C03647=1188.648,139.249,-53.696,-178.416,6.243,148.660
C03648=1188.653,139.000,-53.675,-178.419,6.241,148.660
C03649=1188.658,138.751,-53.655,-178.422,6.239,148.661
C03650=1188.662,138.502,-53.634,-178.424,6.238,148.661
C03651=1188.667,138.252,-53.615,-178.427,6.237,148.662
C03652=1188.672,138.003,-53.594,-178.430,6.235,148.662
C03653=1188.676,137.754,-53.573,-178.432,6.233,148.663
C03654=1188.681,137.505,-53.553,-178.435,6.232,148.663
C03655=1188.686,137.256,-53.532,-178.438,6.231,148.664
C03656=1188.691,137.006,-53.512,-178.440,6.229,148.664
C03657=1188.696,136.758,-53.492,-178.443,6.227,148.664
C03658=1188.700,136.509,-53.472,-178.445,6.226,148.665
C03659=1188.705,136.260,-53.451,-178.448,6.225,148.665
C03660=1188.710,136.010,-53.431,-178.451,6.223,148.666
C03661=1188.714,135.761,-53.411,-178.453,6.222,148.666
C03662=1188.719,135.512,-53.390,-178.456,6.220,148.667
C03663=1188.724,135.262,-53.370,-178.459,6.219,148.667
C03664=1188.729,135.013,-53.350,-178.462,6.217,148.668
C03665=1188.733,134.764,-53.329,-178.464,6.216,148.668
C03666=1188.738,134.515,-53.309,-178.467,6.215,148.668
C03667=1188.744,134.266,-53.289,-178.470,6.213,148.669
C03668=1188.748,134.017,-53.269,-178.472,6.212,148.669
C03669=1188.753,133.768,-53.249,-178.475,6.210,148.670
C03670=1188.757,133.519,-53.229,-178.477,6.209,148.670
C03671=1188.762,133.270,-53.208,-178.480,6.207,148.671
C03672=1188.768,133.001,-53.187,-178.483,6.206,148.671
C03673=1188.772,132.733,-53.165,-178.486,6.205,148.672
C03674=1188.778,132.464,-53.143,-178.488,6.203,148.672
C03675=1188.783,132.195,-53.122,-178.491,6.201,148.673
C03676=1188.787,131.946,-53.102,-178.494,6.200,148.673
C03677=1188.793,131.696,-53.082,-178.497,6.198,148.674
C03678=1188.797,131.447,-53.061,-178.499,6.197,148.674
C03679=1188.802,131.199,-53.042,-178.502,6.196,148.675
C03680=1188.807,130.950,-53.022,-178.505,6.194,148.675
C03681=1188.811,130.701,-53.001,-178.507,6.193,148.675
C03682=1188.816,130.451,-52.981,-178.510,6.191,148.676
C03683=1188.820,130.202,-52.961,-178.513,6.190,148.676
C03684=1188.825,129.953,-52.941,-178.515,6.189,148.677
C03685=1188.831,129.704,-52.922,-178.518,6.187,148.677
C03686=1188.836,129.455,-52.901,-178.521,6.186,148.678
C03687=1188.840,129.205,-52.882,-178.523,6.185,148.678
C03688=1188.845,128.956,-52.861,-178.526,6.183,148.679
C03689=1188.850,128.707,-52.842,-178.529,6.181,148.679
C03690=1188.855,128.458,-52.821,-178.531,6.181,148.680
C03691=1188.859,128.209,-52.802,-178.534,6.179,148.680
C03692=1188.864,127.959,-52.782,-178.537,6.177,148.680
C03693=1188.869,127.710,-52.762,-178.539,6.177,148.681
C03694=1188.874,127.461,-52.743,-178.542,6.175,148.681
C03695=1188.878,127.212,-52.722,-178.545,6.173,148.682
C03696=1188.883,126.963,-52.702,-178.547,6.172,148.682
C03697=1188.888,126.713,-52.683,-178.550,6.171,148.683
C03698=1188.893,126.465,-52.663,-178.553,6.169,148.683
C03699=1188.898,126.215,-52.643,-178.555,6.168,148.684
C03700=1188.902,125.966,-52.624,-178.558,6.167,148.684
C03701=1188.907,125.717,-52.603,-178.561,6.165,148.685
C03702=1188.912,125.468,-52.584,-178.563,6.164,148.685
C03703=1188.916,125.219,-52.565,-178.566,6.163,148.686
C03704=1188.921,124.970,-52.544,-178.569,6.161,148.686
C03705=1188.926,124.721,-52.525,-178.571,6.160,148.686
C03706=1188.931,124.471,-52.505,-178.573,6.158,148.687
C03707=1188.935,124.222,-52.486,-178.576,6.158,148.688
C03708=1188.940,123.973,-52.465,-178.579,6.156,148.688
C03709=1188.945,123.724,-52.446,-178.581,6.154,148.688
C03710=1188.950,123.474,-52.427,-178.584,6.154,148.689
C03711=1188.955,123.225,-52.407,-178.587,6.152,148.689
C03712=1188.960,122.976,-52.388,-178.589,6.150,148.690
C03713=1188.964,122.727,-52.367,-178.592,6.150,148.690
C03714=1188.968,122.478,-52.348,-178.595,6.148,148.691
C03715=1188.974,122.229,-52.329,-178.597,6.146,148.691
C03716=1188.979,121.979,-52.309,-178.600,6.145,148.692
C03717=1188.983,121.730,-52.290,-178.603,6.144,148.692
C03718=1188.989,121.481,-52.270,-178.605,6.143,148.693
C03719=1188.993,121.232,-52.250,-178.608,6.141,148.693
C03720=1188.997,120.983,-52.231,-178.611,6.140,148.694
C03721=1189.002,120.734,-52.212,-178.613,6.139,148.694
C03722=1189.007,120.484,-52.192,-178.616,6.137,148.695
C03723=1189.013,120.235,-52.173,-178.618,6.136,148.695
C03724=1189.017,119.986,-52.153,-178.621,6.135,148.695
C03725=1189.022,119.736,-52.133,-178.624,6.133,148.696
C03726=1189.027,119.488,-52.115,-178.626,6.132,148.696
C03727=1189.031,119.238,-52.095,-178.629,6.131,148.697
C03728=1189.036,118.989,-52.075,-178.632,6.129,148.697
C03729=1189.041,118.740,-52.056,-178.634,6.128,148.698
C03730=1189.045,118.490,-52.037,-178.637,6.126,148.698
C03731=1189.051,118.242,-52.018,-178.639,6.126,148.699
C03732=1189.056,117.992,-51.998,-178.642,6.124,148.699
C03733=1189.060,117.742,-51.978,-178.645,6.122,148.700
C03734=1189.065,117.494,-51.960,-178.647,6.122,148.700
C03735=1189.070,117.244,-51.940,-178.650,6.120,148.701
C03736=1189.075,116.995,-51.921,-178.652,6.119,148.701
C03737=1189.080,116.746,-51.901,-178.655,6.118,148.702
C03738=1189.084,116.497,-51.882,-178.658,6.116,148.702
C03739=1189.089,116.248,-51.863,-178.661,6.115,148.703
C03740=1189.094,115.999,-51.843,-178.663,6.114,148.703
C03741=1189.098,115.750,-51.824,-178.666,6.113,148.704
C03742=1189.103,115.500,-51.805,-178.669,6.111,148.704
C03743=1189.109,115.251,-51.785,-178.671,6.110,148.705
C03744=1189.113,115.002,-51.766,-178.674,6.109,148.705
C03745=1189.118,114.752,-51.748,-178.677,6.107,148.706
C03746=1189.123,114.503,-51.728,-178.679,6.106,148.706
C03747=1189.128,114.254,-51.709,-178.682,6.105,148.707
C03748=1189.132,114.005,-51.690,-178.684,6.104,148.707
C03749=1189.138,113.756,-51.670,-178.687,6.102,148.708
C03750=1189.142,113.507,-51.651,-178.690,6.102,148.708
C03751=1189.147,113.257,-51.633,-178.692,6.100,148.709
C03752=1189.152,113.008,-51.613,-178.695,6.098,148.709
C03753=1189.157,112.759,-51.594,-178.698,6.098,148.710
C03754=1189.161,112.509,-51.575,-178.700,6.096,148.710
C03755=1189.166,112.261,-51.556,-178.702,6.095,148.710
C03756=1189.171,112.011,-51.537,-178.706,6.094,148.711
C03757=1189.176,111.762,-51.518,-178.708,6.093,148.712
C03758=1189.180,111.513,-51.499,-178.711,6.091,148.712
C03759=1189.186,111.263,-51.480,-178.714,6.090,148.713
C03760=1189.190,111.014,-51.461,-178.716,6.089,148.713
C03761=1189.195,110.765,-51.442,-178.719,6.087,148.714
C03762=1189.199,110.516,-51.423,-178.721,6.086,148.714
C03763=1189.205,110.266,-51.404,-178.724,6.085,148.715
C03764=1189.210,110.018,-51.386,-178.726,6.084,148.715
C03765=1189.214,109.768,-51.366,-178.729,6.082,148.715
C03766=1189.219,109.519,-51.348,-178.732,6.082,148.716
C03767=1189.224,109.269,-51.328,-178.734,6.080,148.717
C03768=1189.229,109.021,-51.310,-178.737,6.079,148.717
C03769=1189.234,108.771,-51.291,-178.740,6.078,148.718
C03770=1189.238,108.522,-51.272,-178.742,6.076,148.718
C03771=1189.244,108.273,-51.253,-178.745,6.075,148.719
C03772=1189.248,108.023,-51.234,-178.748,6.074,148.719
C03773=1189.253,107.774,-51.215,-178.750,6.073,148.720
C03774=1189.258,107.525,-51.197,-178.753,6.071,148.720
C03775=1189.263,107.276,-51.177,-178.755,6.070,148.720
C03776=1189.268,107.007,-51.158,-178.758,6.069,148.721
C03777=1189.273,106.739,-51.137,-178.762,6.068,148.722
C03778=1189.279,106.470,-51.117,-178.764,6.067,148.722
C03779=1189.284,106.203,-51.097,-178.767,6.065,148.723
C03780=1189.289,105.952,-51.078,-178.770,6.064,148.723
C03781=1189.293,105.704,-51.059,-178.772,6.063,148.724
C03782=1189.297,105.454,-51.041,-178.775,6.061,148.724
C03783=1189.303,105.205,-51.021,-178.777,6.060,148.725
C03784=1189.308,104.956,-51.003,-178.780,6.059,148.725
C03785=1189.312,104.706,-50.984,-178.782,6.058,148.726
C03786=1189.317,104.457,-50.966,-178.786,6.057,148.726
C03787=1189.322,104.208,-50.948,-178.788,6.056,148.727
C03788=1189.327,103.958,-50.928,-178.791,6.054,148.727
C03789=1189.332,103.709,-50.910,-178.793,6.053,148.728
C03790=1189.337,103.461,-50.892,-178.796,6.052,148.728
C03791=1189.342,103.210,-50.873,-178.798,6.051,148.729
C03792=1189.346,102.962,-50.854,-178.801,6.049,148.729
C03793=1189.351,102.713,-50.836,-178.804,6.049,148.730
C03794=1189.356,102.463,-50.817,-178.806,6.047,148.730
C03795=1189.361,102.214,-50.798,-178.809,6.046,148.731
C03796=1189.366,101.965,-50.780,-178.812,6.045,148.731
C03797=1189.371,101.715,-50.761,-178.814,6.044,148.732
C03798=1189.375,101.466,-50.743,-178.817,6.042,148.732
C03799=1189.380,101.217,-50.725,-178.819,6.041,148.733
C03800=1189.386,100.967,-50.706,-178.822,6.040,148.733
C03801=1189.390,100.718,-50.687,-178.824,6.039,148.734
C03802=1189.395,100.469,-50.669,-178.828,6.038,148.735
C03803=1189.400,100.220,-50.651,-178.830,6.037,148.735
C03804=1189.404,99.970,-50.631,-178.833,6.036,148.736
C03805=1189.409,99.721,-50.613,-178.835,6.035,148.736
C03806=1189.414,99.472,-50.595,-178.838,6.033,148.736
C03807=1189.419,99.223,-50.577,-178.840,6.032,148.737
C03808=1189.424,98.973,-50.558,-178.843,6.031,148.737
C03809=1189.429,98.724,-50.540,-178.846,6.030,148.738
C03810=1189.434,98.475,-50.522,-178.849,6.028,148.739
C03811=1189.439,98.226,-50.504,-178.851,6.028,148.739
C03812=1189.443,97.976,-50.485,-178.854,6.026,148.740
C03813=1189.448,97.727,-50.466,-178.856,6.025,148.740
C03814=1189.453,97.478,-50.448,-178.859,6.024,148.741
C03815=1189.458,97.229,-50.430,-178.861,6.023,148.741
C03816=1189.462,96.979,-50.412,-178.864,6.022,148.742
C03817=1189.467,96.729,-50.394,-178.867,6.020,148.742
C03818=1189.472,96.481,-50.375,-178.869,6.020,148.743
C03819=1189.478,96.231,-50.357,-178.872,6.018,148.743
C03820=1189.483,95.982,-50.339,-178.875,6.018,148.744
C03821=1189.487,95.732,-50.320,-178.877,6.016,148.744
C03822=1189.492,95.483,-50.302,-178.880,6.015,148.745
C03823=1189.497,95.234,-50.284,-178.883,6.014,148.745
C03824=1189.502,94.985,-50.266,-178.885,6.013,148.746
C03825=1189.507,94.736,-50.248,-178.888,6.011,148.746
C03826=1189.512,94.485,-50.229,-178.891,6.011,148.747
C03827=1189.516,94.237,-50.211,-178.893,6.010,148.747
C03828=1189.521,93.988,-50.193,-178.896,6.008,148.748
C03829=1189.526,93.739,-50.175,-178.898,6.008,148.748
C03830=1189.531,93.489,-50.157,-178.901,6.006,148.749
C03831=1189.536,93.240,-50.139,-178.903,6.005,148.750
C03832=1189.540,92.990,-50.121,-178.906,6.003,148.750
C03833=1189.545,92.741,-50.103,-178.909,6.003,148.751
C03834=1189.550,92.492,-50.085,-178.911,6.001,148.751
C03835=1189.555,92.243,-50.067,-178.914,6.001,148.752
C03836=1189.560,91.994,-50.049,-178.916,6.000,148.752
C03837=1189.565,91.744,-50.031,-178.919,5.998,148.753
C03838=1189.570,91.495,-50.013,-178.922,5.997,148.753
C03839=1189.574,91.245,-49.994,-178.925,5.996,148.754
C03840=1189.579,90.996,-49.977,-178.927,5.995,148.754
C03841=1189.584,90.746,-49.959,-178.930,5.994,148.755
C03842=1189.589,90.497,-49.941,-178.932,5.993,148.755
C03843=1189.594,90.248,-49.923,-178.935,5.992,148.756
C03844=1189.599,89.999,-49.905,-178.938,5.991,148.756
C03845=1189.604,89.750,-49.887,-178.940,5.990,148.757
C03846=1189.609,89.501,-49.869,-178.943,5.988,148.757
C03847=1189.614,89.251,-49.851,-178.945,5.988,148.758
C03848=1189.618,89.002,-49.833,-178.948,5.986,148.758
C03849=1189.623,88.752,-49.816,-178.951,5.985,148.759
C03850=1189.628,88.503,-49.798,-178.953,5.985,148.760
C03851=1189.633,88.253,-49.780,-178.956,5.983,148.760
C03852=1189.638,88.004,-49.762,-178.958,5.982,148.761
C03853=1189.643,87.755,-49.744,-178.961,5.981,148.761
C03854=1189.648,87.506,-49.726,-178.964,5.980,148.762
C03855=1189.653,87.256,-49.708,-178.966,5.979,148.762
C03856=1189.658,87.007,-49.690,-178.969,5.978,148.763
C03857=1189.663,86.758,-49.672,-178.972,5.977,148.763
C03858=1189.668,86.509,-49.654,-178.974,5.975,148.764
C03859=1189.672,86.259,-49.638,-178.977,5.975,148.765
C03860=1189.677,86.010,-49.620,-178.979,5.974,148.765
C03861=1189.682,85.761,-49.602,-178.982,5.973,148.766
C03862=1189.687,85.512,-49.584,-178.984,5.972,148.766
C03863=1189.692,85.262,-49.567,-178.988,5.970,148.767
C03864=1189.697,85.013,-49.549,-178.990,5.969,148.767
C03865=1189.702,84.763,-49.531,-178.992,5.969,148.768
C03866=1189.707,84.514,-49.513,-178.996,5.967,148.768
C03867=1189.711,84.265,-49.496,-178.998,5.967,148.769
C03868=1189.716,84.016,-49.478,-179.001,5.965,148.769
C03869=1189.721,83.766,-49.460,-179.003,5.964,148.770
C03870=1189.726,83.517,-49.443,-179.006,5.964,148.771
C03871=1189.731,83.267,-49.425,-179.008,5.962,148.771
C03872=1189.736,83.018,-49.408,-179.011,5.961,148.772
C03873=1189.741,82.769,-49.390,-179.013,5.961,148.772
C03874=1189.745,82.520,-49.372,-179.016,5.959,148.773
C03875=1189.751,82.270,-49.355,-179.018,5.958,148.773
C03876=1189.756,82.021,-49.337,-179.022,5.957,148.774
C03877=1189.760,81.771,-49.320,-179.024,5.956,148.774
C03878=1189.765,81.522,-49.302,-179.026,5.955,148.775
C03879=1189.770,81.273,-49.284,-179.029,5.954,148.775
C03880=1189.775,81.004,-49.266,-179.032,5.953,148.776
C03881=1189.780,80.736,-49.246,-179.035,5.952,148.777
C03882=1189.786,80.468,-49.228,-179.038,5.951,148.777
C03883=1189.791,80.199,-49.210,-179.040,5.950,148.778
C03884=1189.796,79.950,-49.192,-179.043,5.949,148.778
C03885=1189.801,79.700,-49.175,-179.046,5.947,148.779
C03886=1189.805,79.451,-49.157,-179.048,5.947,148.779
C03887=1189.811,79.201,-49.140,-179.050,5.946,148.780
C03888=1189.815,78.952,-49.122,-179.054,5.944,148.780
C03889=1189.821,78.702,-49.105,-179.056,5.944,148.781
C03890=1189.825,78.453,-49.087,-179.058,5.943,148.782
C03891=1189.830,78.204,-49.070,-179.062,5.942,148.782
C03892=1189.836,77.955,-49.052,-179.064,5.941,148.783
C03893=1189.840,77.706,-49.036,-179.066,5.940,148.783
C03894=1189.845,77.456,-49.018,-179.069,5.939,148.784
C03895=1189.850,77.207,-49.000,-179.072,5.938,148.784
C03896=1189.855,76.957,-48.984,-179.074,5.937,148.785
C03897=1189.860,76.708,-48.966,-179.077,5.936,148.785
C03898=1189.865,76.458,-48.949,-179.079,5.935,148.786
C03899=1189.869,76.209,-48.931,-179.082,5.934,148.787
C03900=1189.875,75.960,-48.914,-179.085,5.933,148.787
C03901=1189.879,75.711,-48.898,-179.087,5.932,148.788
C03902=1189.884,75.462,-48.880,-179.090,5.931,148.788
C03903=1189.889,75.212,-48.862,-179.093,5.930,148.789
C03904=1189.894,74.962,-48.846,-179.095,5.929,148.789
C03905=1189.899,74.713,-48.828,-179.097,5.928,148.790
C03906=1189.903,74.464,-48.811,-179.101,5.927,148.790
C03907=1189.909,74.215,-48.794,-179.103,5.926,148.791
C03908=1189.914,73.965,-48.776,-179.105,5.925,148.792
C03909=1189.918,73.716,-48.759,-179.109,5.924,148.792
C03910=1189.924,73.466,-48.742,-179.111,5.923,148.793
C03911=1189.928,73.217,-48.726,-179.113,5.923,148.793
C03912=1189.933,72.967,-48.708,-179.116,5.921,148.794
C03913=1189.938,72.719,-48.691,-179.119,5.920,148.794
C03914=1189.943,72.469,-48.674,-179.121,5.920,148.795
C03915=1189.948,72.219,-48.657,-179.124,5.918,148.795
C03916=1189.953,71.970,-48.639,-179.127,5.918,148.796
C03917=1189.957,71.721,-48.623,-179.129,5.917,148.797
C03918=1189.963,71.472,-48.606,-179.132,5.915,148.797
C03919=1189.968,71.222,-48.589,-179.134,5.914,148.798
C03920=1189.973,70.972,-48.572,-179.137,5.914,148.798
C03921=1189.977,70.724,-48.554,-179.140,5.913,148.799
C03922=1189.983,70.474,-48.538,-179.142,5.912,148.799
C03923=1189.987,70.225,-48.521,-179.145,5.911,148.800
C03924=1189.992,69.975,-48.504,-179.147,5.910,148.800
C03925=1189.997,69.726,-48.487,-179.150,5.909,148.801
C03926=1190.003,69.477,-48.470,-179.152,5.908,148.802
C03927=1190.007,69.227,-48.453,-179.155,5.907,148.802
C03928=1190.012,68.977,-48.436,-179.158,5.906,148.803
C03929=1190.017,68.728,-48.419,-179.160,5.905,148.803
C03930=1190.021,68.479,-48.402,-179.163,5.905,148.804
C03931=1190.027,68.230,-48.385,-179.165,5.904,148.804
C03932=1190.031,67.980,-48.368,-179.168,5.902,148.805
C03933=1190.037,67.731,-48.351,-179.171,5.902,148.806
C03934=1190.042,67.482,-48.335,-179.173,5.901,148.806
C03935=1190.046,67.232,-48.318,-179.176,5.900,148.807
C03936=1190.051,66.982,-48.301,-179.178,5.899,148.807
C03937=1190.056,66.733,-48.284,-179.181,5.898,148.808
C03938=1190.062,66.484,-48.267,-179.184,5.898,148.809
C03939=1190.066,66.234,-48.251,-179.186,5.896,148.809
C03940=1190.071,65.985,-48.234,-179.189,5.895,148.810
C03941=1190.077,65.736,-48.217,-179.191,5.894,148.810
C03942=1190.081,65.486,-48.201,-179.194,5.893,148.811
C03943=1190.085,65.237,-48.184,-179.197,5.893,148.811
C03944=1190.091,64.988,-48.167,-179.199,5.892,148.812
C03945=1190.096,64.738,-48.150,-179.202,5.891,148.812
C03946=1190.100,64.489,-48.134,-179.204,5.889,148.813
C03947=1190.105,64.239,-48.116,-179.207,5.889,148.814
C03948=1190.111,63.990,-48.100,-179.210,5.888,148.814
C03949=1190.115,63.741,-48.083,-179.212,5.887,148.815
C03950=1190.120,63.491,-48.066,-179.215,5.886,148.815
C03951=1190.126,63.242,-48.051,-179.217,5.885,148.816
C03952=1190.130,62.992,-48.034,-179.220,5.885,148.816
C03953=1190.136,62.743,-48.017,-179.223,5.883,148.817
C03954=1190.140,62.494,-48.000,-179.225,5.882,148.818
C03955=1190.145,62.244,-47.984,-179.228,5.882,148.818
C03956=1190.150,61.995,-47.967,-179.230,5.881,148.819
C03957=1190.155,61.745,-47.950,-179.233,5.880,148.819
C03958=1190.160,61.496,-47.933,-179.236,5.879,148.820
C03959=1190.165,61.247,-47.918,-179.238,5.878,148.820
C03960=1190.170,60.997,-47.901,-179.241,5.878,148.821
C03961=1190.175,60.748,-47.884,-179.244,5.876,148.822
C03962=1190.180,60.498,-47.868,-179.246,5.875,148.822
C03963=1190.184,60.249,-47.851,-179.249,5.875,148.823
C03964=1190.190,60.000,-47.835,-179.251,5.874,148.823
C03965=1190.194,59.750,-47.819,-179.254,5.873,148.824
C03966=1190.200,59.501,-47.802,-179.257,5.872,148.825
C03967=1190.204,59.252,-47.785,-179.259,5.871,148.825
C03968=1190.209,59.001,-47.769,-179.261,5.871,148.826
C03969=1190.214,58.753,-47.753,-179.264,5.870,148.826
C03970=1190.219,58.503,-47.736,-179.267,5.869,148.827
C03971=1190.225,58.254,-47.719,-179.269,5.868,148.827
C03972=1190.229,58.004,-47.703,-179.272,5.867,148.828
C03973=1190.235,57.755,-47.687,-179.274,5.867,148.829
C03974=1190.239,57.506,-47.670,-179.277,5.865,148.829
C03975=1190.244,57.256,-47.654,-179.280,5.864,148.830
C03976=1190.249,57.007,-47.638,-179.282,5.864,148.830
C03977=1190.254,56.757,-47.621,-179.285,5.863,148.831
C03978=1190.259,56.508,-47.605,-179.288,5.862,148.831
C03979=1190.264,56.258,-47.589,-179.290,5.861,148.832
C03980=1190.269,56.009,-47.572,-179.292,5.860,148.832
C03981=1190.274,55.759,-47.556,-179.295,5.860,148.833
C03982=1190.279,55.510,-47.540,-179.298,5.859,148.834
C03983=1190.284,55.260,-47.524,-179.300,5.857,148.834
C03984=1190.289,54.993,-47.506,-179.303,5.857,148.835
C03985=1190.294,54.723,-47.489,-179.306,5.856,148.836
C03986=1190.300,54.455,-47.471,-179.309,5.855,148.836
C03987=1190.305,54.187,-47.454,-179.311,5.854,148.837
C03988=1190.310,53.937,-47.437,-179.314,5.854,148.837
C03989=1190.315,53.688,-47.421,-179.317,5.852,148.838
C03990=1190.320,53.438,-47.405,-179.319,5.852,148.839
C03991=1190.325,53.189,-47.389,-179.322,5.851,148.839
C03992=1190.330,52.939,-47.372,-179.324,5.850,148.840
C03993=1190.335,52.690,-47.357,-179.327,5.850,148.840
C03994=1190.340,52.441,-47.340,-179.330,5.848,148.841
C03995=1190.345,52.191,-47.325,-179.332,5.848,148.842
C03996=1190.349,51.942,-47.308,-179.334,5.847,148.842
C03997=1190.355,51.692,-47.292,-179.337,5.846,148.843
C03998=1190.360,51.443,-47.276,-179.340,5.846,148.843
C03999=1190.365,51.193,-47.260,-179.342,5.844,148.844
C04000=1190.370,50.945,-47.244,-179.345,5.843,148.844
C04001=1190.374,50.694,-47.228,-179.348,5.843,148.845
C04002=1190.380,50.445,-47.212,-179.350,5.842,148.846
C04003=1190.384,50.196,-47.195,-179.352,5.841,148.846
C04004=1190.390,49.946,-47.180,-179.356,5.840,148.847
C04005=1190.394,49.697,-47.163,-179.358,5.839,148.847
C04006=1190.400,49.447,-47.148,-179.360,5.839,148.848
C04007=1190.405,49.199,-47.131,-179.363,5.838,148.849
C04008=1190.409,48.948,-47.115,-179.365,5.837,148.849
C04009=1190.415,48.699,-47.100,-179.368,5.837,148.850
C04010=1190.419,48.450,-47.083,-179.371,5.835,148.850
C04011=1190.424,48.200,-47.068,-179.373,5.835,148.851
C04012=1190.429,47.950,-47.052,-179.376,5.834,148.852
C04013=1190.434,47.702,-47.036,-179.379,5.834,148.852
C04014=1190.439,47.452,-47.020,-179.381,5.833,148.853
C04015=1190.444,47.202,-47.004,-179.383,5.832,148.853
C04016=1190.449,46.953,-46.988,-179.387,5.831,148.854
C04017=1190.455,46.704,-46.972,-179.389,5.830,148.854
C04018=1190.459,46.454,-46.957,-179.391,5.829,148.855
C04019=1190.464,46.205,-46.940,-179.394,5.829,148.856
C04020=1190.468,45.955,-46.925,-179.396,5.828,148.856
C04021=1190.474,45.706,-46.909,-179.399,5.827,148.857
C04022=1190.479,45.456,-46.894,-179.402,5.826,148.858
C04023=1190.484,45.207,-46.877,-179.404,5.825,148.858
C04024=1190.489,44.957,-46.861,-179.407,5.825,148.859
C04025=1190.494,44.708,-46.846,-179.409,5.824,148.859
C04026=1190.499,44.458,-46.830,-179.412,5.823,148.860
C04027=1190.504,44.210,-46.814,-179.414,5.823,148.860
C04028=1190.509,43.960,-46.799,-179.417,5.821,148.861
C04029=1190.514,43.710,-46.783,-179.420,5.821,148.862
C04030=1190.519,43.461,-46.767,-179.422,5.820,148.862
C04031=1190.525,43.211,-46.751,-179.425,5.820,148.863
C04032=1190.528,42.962,-46.735,-179.427,5.819,148.863
C04033=1190.534,42.713,-46.720,-179.430,5.818,148.864
C04034=1190.539,42.463,-46.704,-179.432,5.818,148.865
C04035=1190.544,42.213,-46.688,-179.435,5.816,148.865
C04036=1190.548,41.964,-46.673,-179.438,5.815,148.866
C04037=1190.554,41.715,-46.658,-179.440,5.815,148.867
C04038=1190.559,41.465,-46.642,-179.442,5.814,148.867
C04039=1190.564,41.215,-46.626,-179.445,5.813,148.868
C04040=1190.568,40.967,-46.610,-179.448,5.813,148.868
C04041=1190.574,40.717,-46.595,-179.450,5.812,148.869
C04042=1190.579,40.467,-46.579,-179.453,5.811,148.869
C04043=1190.584,40.218,-46.563,-179.456,5.810,148.870
C04044=1190.589,39.969,-46.548,-179.458,5.810,148.871
C04045=1190.593,39.719,-46.532,-179.461,5.809,148.871
C04046=1190.599,39.469,-46.517,-179.463,5.808,148.872
C04047=1190.604,39.220,-46.501,-179.466,5.808,148.873
C04048=1190.609,38.971,-46.486,-179.468,5.807,148.873
C04049=1190.614,38.721,-46.470,-179.471,5.806,148.874
C04050=1190.619,38.471,-46.455,-179.474,5.805,148.874
C04051=1190.624,38.222,-46.440,-179.476,5.804,148.875
C04052=1190.629,37.973,-46.424,-179.479,5.804,148.875
C04053=1190.634,37.723,-46.408,-179.481,5.803,148.876
C04054=1190.638,37.473,-46.393,-179.483,5.802,148.877
C04055=1190.644,37.224,-46.378,-179.486,5.802,148.877
C04056=1190.649,36.975,-46.362,-179.489,5.801,148.878
C04057=1190.654,36.726,-46.347,-179.491,5.801,148.879
C04058=1190.659,36.475,-46.331,-179.494,5.800,148.879
C04059=1190.664,36.226,-46.315,-179.497,5.799,148.880
C04060=1190.669,35.977,-46.300,-179.499,5.798,148.880
C04061=1190.674,35.728,-46.285,-179.502,5.797,148.881
C04062=1190.679,35.478,-46.270,-179.504,5.797,148.882
C04063=1190.684,35.228,-46.254,-179.507,5.796,148.882
C04064=1190.689,34.978,-46.239,-179.509,5.795,148.883
C04065=1190.694,34.729,-46.224,-179.512,5.795,148.883
C04066=1190.699,34.480,-46.208,-179.514,5.794,148.884
C04067=1190.704,34.231,-46.193,-179.517,5.794,148.885
C04068=1190.709,33.981,-46.177,-179.520,5.792,148.885
C04069=1190.713,33.732,-46.162,-179.522,5.792,148.886
C04070=1190.719,33.482,-46.147,-179.525,5.791,148.886
C04071=1190.724,33.232,-46.132,-179.527,5.790,148.887
C04072=1190.729,32.983,-46.117,-179.530,5.790,148.888
C04073=1190.734,32.734,-46.101,-179.532,5.789,148.888
C04074=1190.738,32.484,-46.086,-179.535,5.788,148.889
C04075=1190.744,32.234,-46.070,-179.537,5.788,148.889
C04076=1190.749,31.985,-46.056,-179.540,5.787,148.890
C04077=1190.754,31.735,-46.041,-179.542,5.787,148.891
C04078=1190.759,31.486,-46.026,-179.545,5.786,148.891
C04079=1190.764,31.237,-46.010,-179.547,5.785,148.892
C04080=1190.769,30.988,-45.995,-179.551,5.784,148.893
C04081=1190.774,30.737,-45.980,-179.553,5.783,148.893
C04082=1190.779,30.488,-45.965,-179.555,5.783,148.894
C04083=1190.784,30.239,-45.949,-179.558,5.782,148.894
C04084=1190.789,29.989,-45.935,-179.561,5.782,148.895
C04085=1190.794,29.739,-45.919,-179.563,5.781,148.895
C04086=1190.799,29.490,-45.904,-179.565,5.780,148.896
C04087=1190.804,29.241,-45.889,-179.568,5.780,148.897
C04088=1190.810,28.972,-45.873,-179.571,5.779,148.898
C04089=1190.815,28.703,-45.857,-179.574,5.778,148.898
C04090=1190.821,28.434,-45.841,-179.576,5.777,148.899
C04091=1190.826,28.166,-45.824,-179.579,5.777,148.899
C04092=1190.831,27.916,-45.810,-179.581,5.776,148.900
C04093=1190.836,27.667,-45.795,-179.584,5.776,148.901
C04094=1190.841,27.418,-45.779,-179.587,5.775,148.901
C04095=1190.845,27.167,-45.765,-179.589,5.774,148.902
C04096=1190.851,26.918,-45.749,-179.591,5.774,148.902
C04097=1190.855,26.669,-45.734,-179.594,5.773,148.903
C04098=1190.860,26.419,-45.720,-179.596,5.772,148.904
C04099=1190.866,26.170,-45.704,-179.599,5.772,148.904
C04100=1190.871,25.920,-45.690,-179.602,5.770,148.905
C04101=1190.876,25.670,-45.674,-179.605,5.770,148.906
C04102=1190.881,25.421,-45.660,-179.607,5.769,148.906
C04103=1190.886,25.172,-45.645,-179.610,5.769,148.907
C04104=1190.891,24.922,-45.629,-179.612,5.768,148.907
C04105=1190.896,24.673,-45.615,-179.614,5.767,148.908
C04106=1190.901,24.423,-45.600,-179.617,5.767,148.909
C04107=1190.906,24.173,-45.585,-179.620,5.766,148.909
C04108=1190.911,23.924,-45.570,-179.622,5.766,148.910
C04109=1190.916,23.675,-45.556,-179.625,5.765,148.910
C04110=1190.921,23.425,-45.540,-179.627,5.764,148.911
C04111=1190.926,23.175,-45.526,-179.630,5.764,148.912
C04112=1190.931,22.926,-45.511,-179.632,5.763,148.912
C04113=1190.937,22.676,-45.496,-179.635,5.762,148.913
C04114=1190.941,22.427,-45.481,-179.637,5.762,148.914
C04115=1190.946,22.178,-45.467,-179.640,5.761,148.914
C04116=1190.951,21.928,-45.453,-179.642,5.761,148.915
C04117=1190.957,21.678,-45.437,-179.645,5.760,148.915
C04118=1190.962,21.429,-45.423,-179.647,5.760,148.916
C04119=1190.966,21.180,-45.408,-179.650,5.759,148.917
C04120=1190.972,20.930,-45.393,-179.652,5.758,148.917
C04121=1190.977,20.681,-45.378,-179.655,5.758,148.918
C04122=1190.982,20.431,-45.364,-179.657,5.757,148.919
C04123=1190.987,20.181,-45.349,-179.660,5.757,148.919
C04124=1190.992,19.932,-45.334,-179.662,5.756,148.920
C04125=1190.997,19.682,-45.320,-179.665,5.755,148.920
C04126=1191.002,19.432,-45.305,-179.668,5.754,148.921
C04127=1191.006,19.183,-45.290,-179.671,5.754,148.922
C04128=1191.011,18.933,-45.276,-179.673,5.753,148.922
C04129=1191.017,18.684,-45.260,-179.676,5.752,148.923
C04130=1191.022,18.434,-45.246,-179.678,5.752,148.924
C04131=1191.027,18.185,-45.232,-179.680,5.751,148.924
C04132=1191.032,17.936,-45.218,-179.683,5.750,148.925
C04133=1191.037,17.687,-45.203,-179.686,5.750,148.925
C04134=1191.043,17.437,-45.188,-179.688,5.749,148.926
C04135=1191.048,17.187,-45.174,-179.691,5.749,148.927
C04136=1191.052,16.938,-45.159,-179.693,5.748,148.927
C04137=1191.057,16.688,-45.145,-179.696,5.748,148.928
C04138=1191.062,16.438,-45.130,-179.698,5.747,148.929
C04139=1191.067,16.189,-45.116,-179.701,5.746,148.929
C04140=1191.072,15.940,-45.101,-179.703,5.746,148.930
C04141=1191.077,15.689,-45.086,-179.706,5.745,148.930
C04142=1191.083,15.440,-45.072,-179.709,5.745,148.931
C04143=1191.088,15.191,-45.058,-179.711,5.744,148.932
C04144=1191.093,14.942,-45.043,-179.713,5.743,148.932
C04145=1191.098,14.692,-45.029,-179.716,5.743,148.933
C04146=1191.102,14.442,-45.014,-179.719,5.742,148.934
C04147=1191.107,14.193,-45.000,-179.721,5.741,148.934
C04148=1191.112,13.943,-44.986,-179.724,5.741,148.935
C04149=1191.117,13.694,-44.971,-179.726,5.740,148.935
C04150=1191.123,13.444,-44.956,-179.729,5.740,148.936
C04151=1191.128,13.195,-44.942,-179.731,5.739,148.937
C04152=1191.133,12.945,-44.928,-179.734,5.739,148.937
C04153=1191.138,12.695,-44.913,-179.736,5.738,148.938
C04154=1191.143,12.446,-44.899,-179.739,5.738,148.939
C04155=1191.148,12.196,-44.885,-179.741,5.737,148.939
C04156=1191.154,11.947,-44.871,-179.744,5.736,148.940
C04157=1191.158,11.698,-44.856,-179.746,5.736,148.940
C04158=1191.163,11.448,-44.842,-179.748,5.736,148.941
C04159=1191.168,11.198,-44.827,-179.751,5.735,148.942
C04160=1191.173,10.949,-44.813,-179.753,5.735,148.942
C04161=1191.178,10.699,-44.799,-179.756,5.734,148.943
C04162=1191.184,10.450,-44.785,-179.759,5.734,148.944
C04163=1191.189,10.200,-44.771,-179.761,5.733,148.944
C04164=1191.194,9.951,-44.756,-179.763,5.732,148.945
C04165=1191.199,9.701,-44.742,-179.766,5.732,148.945
C04166=1191.204,9.451,-44.728,-179.769,5.731,148.946
C04167=1191.209,9.202,-44.714,-179.771,5.731,148.947
C04168=1191.214,8.952,-44.700,-179.774,5.730,148.947
C04169=1191.219,8.703,-44.685,-179.776,5.730,148.948
C04170=1191.224,8.453,-44.671,-179.779,5.729,148.949
C04171=1191.229,8.204,-44.657,-179.781,5.728,148.949
C04172=1191.234,7.954,-44.643,-179.784,5.728,148.950
C04173=1191.239,7.705,-44.629,-179.786,5.727,148.950
C04174=1191.244,7.455,-44.614,-179.789,5.727,148.951
C04175=1191.249,7.205,-44.600,-179.791,5.726,148.952
C04176=1191.255,6.956,-44.586,-179.794,5.725,148.952
C04177=1191.260,6.706,-44.572,-179.796,5.725,148.953
C04178=1191.264,6.457,-44.558,-179.799,5.724,148.954
C04179=1191.269,6.207,-44.544,-179.801,5.724,148.954
C04180=1191.275,5.958,-44.530,-179.804,5.723,148.955
C04181=1191.279,5.709,-44.516,-179.807,5.723,148.956
C04182=1191.284,5.459,-44.502,-179.809,5.722,148.956
C04183=1191.290,5.208,-44.488,-179.811,5.721,148.957
C04184=1191.295,4.959,-44.474,-179.814,5.721,148.957
C04185=1191.300,4.710,-44.460,-179.816,5.721,148.958
C04186=1191.305,4.460,-44.445,-179.819,5.721,148.959
C04187=1191.310,4.211,-44.432,-179.821,5.720,148.959
C04188=1191.315,3.962,-44.418,-179.824,5.719,148.960
C04189=1191.320,3.712,-44.404,-179.826,5.719,148.961
C04190=1191.325,3.462,-44.390,-179.829,5.718,148.961
C04191=1191.331,3.213,-44.376,-179.831,5.718,148.962
C04192=1191.336,2.943,-44.361,-179.834,5.717,148.963
C04193=1191.341,2.674,-44.345,-179.837,5.717,148.963
C04194=1191.347,2.405,-44.330,-179.839,5.716,148.964
C04195=1191.353,2.136,-44.316,-179.842,5.716,148.964
C04196=1191.358,1.887,-44.302,-179.844,5.715,148.965
C04197=1191.362,1.637,-44.289,-179.847,5.715,148.966
C04198=1191.368,1.388,-44.275,-179.850,5.714,148.967
C04199=1191.373,1.138,-44.260,-179.852,5.714,148.967
C04200=1191.378,0.888,-44.246,-179.854,5.713,148.968
C04201=1191.383,0.639,-44.234,-179.857,5.712,148.968
C04202=1191.388,0.389,-44.219,-179.860,5.712,148.969
C04203=1191.393,0.139,-44.205,-179.862,5.711,148.970
C04204=1191.398,-0.110,-44.191,-179.865,5.710,148.970
C04205=1191.404,-0.360,-44.177,-179.867,5.710,148.971
C04206=1191.408,-0.609,-44.164,-179.870,5.709,148.972
C04207=1191.413,-0.858,-44.150,-179.872,5.709,148.972
C04208=1191.419,-1.109,-44.136,-179.875,5.708,148.973
C04209=1191.424,-1.358,-44.122,-179.877,5.708,148.973
C04210=1191.428,-1.607,-44.109,-179.879,5.708,148.974
C04211=1191.434,-1.857,-44.095,-179.882,5.708,148.975
C04212=1191.439,-2.106,-44.081,-179.885,5.707,148.975
C04213=1191.443,-2.356,-44.068,-179.887,5.706,148.976
C04214=1191.449,-2.606,-44.054,-179.890,5.706,148.977
C04215=1191.454,-2.855,-44.040,-179.892,5.705,148.977
C04216=1191.459,-3.105,-44.026,-179.895,5.705,148.978
C04217=1191.464,-3.354,-44.013,-179.897,5.704,148.978
C04218=1191.469,-3.604,-43.999,-179.900,5.703,148.979
C04219=1191.474,-3.854,-43.985,-179.902,5.703,148.980
C04220=1191.479,-4.103,-43.972,-179.904,5.703,148.981
C04221=1191.484,-4.353,-43.958,-179.907,5.702,148.981
C04222=1191.490,-4.602,-43.945,-179.909,5.702,148.982
C04223=1191.494,-4.852,-43.931,-179.912,5.701,148.982
C04224=1191.500,-5.101,-43.918,-179.915,5.701,148.983
C04225=1191.505,-5.351,-43.903,-179.917,5.700,148.984
C04226=1191.510,-5.601,-43.890,-179.919,5.700,148.984
C04227=1191.515,-5.850,-43.877,-179.922,5.699,148.985
C04228=1191.521,-6.100,-43.863,-179.925,5.699,148.986
C04229=1191.525,-6.349,-43.850,-179.927,5.698,148.986
C04230=1191.531,-6.599,-43.836,-179.929,5.698,148.987
C04231=1191.535,-6.848,-43.823,-179.932,5.698,148.987
C04232=1191.541,-7.098,-43.809,-179.934,5.697,148.988
C04233=1191.546,-7.347,-43.795,-179.937,5.697,148.989
C04234=1191.551,-7.597,-43.782,-179.939,5.696,148.989
C04235=1191.556,-7.847,-43.768,-179.942,5.695,148.990
C04236=1191.561,-8.096,-43.756,-179.944,5.695,148.991
C04237=1191.566,-8.346,-43.741,-179.947,5.694,148.991
C04238=1191.571,-8.596,-43.729,-179.950,5.694,148.992
C04239=1191.576,-8.845,-43.714,-179.951,5.694,148.993
C04240=1191.582,-9.095,-43.701,-179.954,5.693,148.993
C04241=1191.586,-9.344,-43.687,-179.957,5.693,148.994
C04242=1191.592,-9.594,-43.674,-179.959,5.693,148.995
C04243=1191.596,-9.844,-43.661,-179.961,5.692,148.995
C04244=1191.602,-10.093,-43.647,-179.964,5.691,148.996
C04245=1191.606,-10.343,-43.634,-179.967,5.691,148.996
C04246=1191.612,-10.592,-43.621,-179.969,5.690,148.997
C04247=1191.616,-10.842,-43.608,-179.971,5.691,148.998
C04248=1191.622,-11.092,-43.594,-179.974,5.690,148.998
C04249=1191.627,-11.341,-43.581,-179.976,5.689,148.999
C04250=1191.632,-11.591,-43.567,-179.979,5.689,149.000
C04251=1191.637,-11.841,-43.555,-179.982,5.688,149.000
C04252=1191.642,-12.090,-43.541,-179.984,5.687,149.001
C04253=1191.647,-12.340,-43.528,-179.986,5.687,149.002
C04254=1191.653,-12.589,-43.514,-179.988,5.687,149.002
C04255=1191.658,-12.838,-43.501,-179.991,5.687,149.003
C04256=1191.663,-13.088,-43.488,-179.994,5.686,149.004
C04257=1191.668,-13.338,-43.475,-179.996,5.686,149.004
C04258=1191.673,-13.588,-43.461,-179.999,5.685,149.005
C04259=1191.678,-13.837,-43.448,179.999,5.685,149.005
C04260=1191.683,-14.087,-43.435,179.996,5.684,149.006
C04261=1191.689,-14.336,-43.422,179.994,5.683,149.007
C04262=1191.693,-14.586,-43.408,179.992,5.684,149.007
C04263=1191.699,-14.835,-43.395,179.989,5.683,149.008
C04264=1191.704,-15.085,-43.382,179.987,5.683,149.009
C04265=1191.709,-15.335,-43.369,179.984,5.682,149.009
C04266=1191.714,-15.584,-43.356,179.982,5.681,149.010
C04267=1191.719,-15.834,-43.342,179.979,5.681,149.011
C04268=1191.724,-16.083,-43.329,179.977,5.681,149.011
C04269=1191.729,-16.333,-43.317,179.974,5.681,149.012
C04270=1191.735,-16.583,-43.303,179.972,5.680,149.012
C04271=1191.740,-16.832,-43.291,179.969,5.679,149.013
C04272=1191.745,-17.082,-43.276,179.967,5.679,149.014
C04273=1191.750,-17.331,-43.264,179.964,5.679,149.014
C04274=1191.755,-17.581,-43.251,179.961,5.678,149.015
C04275=1191.760,-17.831,-43.238,179.960,5.678,149.016
C04276=1191.765,-18.080,-43.225,179.957,5.678,149.016
C04277=1191.770,-18.330,-43.212,179.955,5.677,149.017
C04278=1191.776,-18.580,-43.199,179.952,5.677,149.018
C04279=1191.780,-18.829,-43.186,179.950,5.676,149.018
C04280=1191.785,-19.079,-43.173,179.947,5.675,149.019
C04281=1191.791,-19.328,-43.159,179.945,5.676,149.020
C04282=1191.796,-19.578,-43.147,179.942,5.675,149.020
C04283=1191.801,-19.828,-43.134,179.940,5.675,149.021
C04284=1191.806,-20.077,-43.121,179.938,5.674,149.021
C04285=1191.812,-20.327,-43.108,179.935,5.673,149.022
C04286=1191.816,-20.577,-43.095,179.932,5.673,149.023
C04287=1191.822,-20.826,-43.082,179.930,5.673,149.024
C04288=1191.827,-21.076,-43.069,179.928,5.672,149.024
C04289=1191.832,-21.326,-43.056,179.925,5.672,149.025
C04290=1191.837,-21.575,-43.043,179.923,5.671,149.025
C04291=1191.843,-21.825,-43.030,179.920,5.671,149.026
C04292=1191.847,-22.075,-43.018,179.917,5.671,149.027
C04293=1191.852,-22.324,-43.005,179.916,5.671,149.027
C04294=1191.858,-22.573,-42.992,179.913,5.670,149.028
C04295=1191.863,-22.823,-42.979,179.910,5.670,149.029
C04296=1191.869,-23.093,-42.965,179.908,5.669,149.029
C04297=1191.874,-23.362,-42.950,179.905,5.669,149.030
C04298=1191.879,-23.632,-42.937,179.902,5.668,149.031
C04299=1191.885,-23.901,-42.923,179.900,5.668,149.031
C04300=1191.889,-24.151,-42.910,179.897,5.667,149.032
C04301=1191.895,-24.401,-42.898,179.895,5.668,149.033
C04302=1191.901,-24.651,-42.885,179.893,5.667,149.033
C04303=1191.906,-24.900,-42.872,179.890,5.666,149.034
C04304=1191.910,-25.150,-42.859,179.888,5.666,149.035
C04305=1191.916,-25.399,-42.847,179.885,5.665,149.035
C04306=1191.921,-25.649,-42.834,179.883,5.665,149.036
C04307=1191.926,-25.899,-42.820,179.881,5.665,149.037
C04308=1191.931,-26.148,-42.808,179.878,5.664,149.037
C04309=1191.936,-26.398,-42.795,179.875,5.664,149.038
C04310=1191.941,-26.647,-42.783,179.873,5.664,149.039
C04311=1191.946,-26.897,-42.770,179.871,5.663,149.039
C04312=1191.951,-27.147,-42.758,179.868,5.663,149.040
C04313=1191.956,-27.396,-42.745,179.866,5.663,149.040
C04314=1191.962,-27.646,-42.732,179.863,5.662,149.041
C04315=1191.967,-27.896,-42.719,179.861,5.661,149.042
C04316=1191.972,-28.145,-42.706,179.859,5.662,149.042
C04317=1191.977,-28.394,-42.694,179.856,5.661,149.043
C04318=1191.982,-28.644,-42.682,179.854,5.661,149.044
C04319=1191.988,-28.894,-42.669,179.851,5.660,149.044
C04320=1191.992,-29.144,-42.656,179.849,5.659,149.045
C04321=1191.998,-29.393,-42.643,179.847,5.660,149.046
C04322=1192.003,-29.643,-42.631,179.844,5.659,149.046
C04323=1192.008,-29.893,-42.619,179.841,5.659,149.047
C04324=1192.014,-30.142,-42.606,179.839,5.658,149.047
C04325=1192.018,-30.392,-42.593,179.836,5.658,149.048
C04326=1192.023,-30.641,-42.581,179.834,5.658,149.049
C04327=1192.029,-30.891,-42.569,179.832,5.657,149.050
C04328=1192.034,-31.140,-42.556,179.829,5.657,149.050
C04329=1192.039,-31.390,-42.543,179.827,5.656,149.051
C04330=1192.043,-31.640,-42.530,179.825,5.656,149.051
C04331=1192.049,-31.890,-42.519,179.822,5.656,149.052
C04332=1192.054,-32.139,-42.506,179.819,5.656,149.053
C04333=1192.059,-32.388,-42.493,179.817,5.655,149.054
C04334=1192.065,-32.638,-42.482,179.815,5.654,149.054
C04335=1192.070,-32.888,-42.468,179.813,5.655,149.055
C04336=1192.075,-33.138,-42.455,179.810,5.654,149.055
C04337=1192.080,-33.388,-42.443,179.807,5.654,149.056
C04338=1192.085,-33.637,-42.431,179.805,5.653,149.057
C04339=1192.091,-33.887,-42.418,179.803,5.653,149.057
C04340=1192.096,-34.136,-42.406,179.800,5.653,149.058
C04341=1192.101,-34.386,-42.394,179.798,5.652,149.059
C04342=1192.106,-34.635,-42.381,179.795,5.652,149.059
C04343=1192.111,-34.886,-42.369,179.793,5.651,149.060
C04344=1192.116,-35.135,-42.356,179.791,5.651,149.061
C04345=1192.121,-35.384,-42.344,179.788,5.651,149.061
C04346=1192.127,-35.634,-42.332,179.785,5.650,149.062
C04347=1192.132,-35.884,-42.319,179.783,5.650,149.062
C04348=1192.137,-36.134,-42.307,179.781,5.650,149.063
C04349=1192.142,-36.383,-42.295,179.778,5.650,149.064
C04350=1192.147,-36.632,-42.283,179.776,5.649,149.064
C04351=1192.152,-36.882,-42.271,179.773,5.649,149.065
C04352=1192.157,-37.132,-42.258,179.772,5.649,149.066
C04353=1192.162,-37.382,-42.246,179.769,5.648,149.066
C04354=1192.167,-37.631,-42.233,179.766,5.648,149.067
C04355=1192.173,-37.881,-42.222,179.764,5.647,149.068
C04356=1192.178,-38.130,-42.209,179.762,5.647,149.068
C04357=1192.183,-38.380,-42.197,179.759,5.647,149.069
C04358=1192.188,-38.630,-42.184,179.757,5.646,149.070
C04359=1192.194,-38.880,-42.173,179.754,5.646,149.070
C04360=1192.199,-39.129,-42.160,179.752,5.646,149.071
C04361=1192.204,-39.379,-42.148,179.750,5.645,149.071
C04362=1192.210,-39.628,-42.135,179.747,5.645,149.072
C04363=1192.214,-39.878,-42.124,179.744,5.645,149.073
C04364=1192.219,-40.127,-42.112,179.742,5.645,149.074
C04365=1192.225,-40.377,-42.100,179.740,5.644,149.074
C04366=1192.229,-40.627,-42.087,179.738,5.644,149.075
C04367=1192.235,-40.877,-42.075,179.735,5.643,149.075
C04368=1192.240,-41.127,-42.063,179.733,5.643,149.076
C04369=1192.245,-41.376,-42.050,179.731,5.643,149.077
C04370=1192.250,-41.626,-42.039,179.728,5.642,149.077
C04371=1192.255,-41.875,-42.026,179.725,5.642,149.078
C04372=1192.261,-42.125,-42.015,179.723,5.642,149.079
C04373=1192.266,-42.374,-42.002,179.721,5.642,149.079
C04374=1192.271,-42.624,-41.990,179.718,5.641,149.080
C04375=1192.277,-42.874,-41.978,179.716,5.640,149.081
C04376=1192.281,-43.123,-41.966,179.714,5.641,149.081
C04377=1192.286,-43.373,-41.954,179.711,5.640,149.082
C04378=1192.292,-43.623,-41.942,179.709,5.639,149.082
C04379=1192.297,-43.872,-41.930,179.707,5.640,149.083
C04380=1192.302,-44.122,-41.918,179.704,5.639,149.084
C04381=1192.307,-44.372,-41.907,179.701,5.639,149.085
C04382=1192.312,-44.621,-41.894,179.699,5.638,149.085
C04383=1192.318,-44.871,-41.882,179.697,5.638,149.086
C04384=1192.323,-45.121,-41.870,179.694,5.638,149.086
C04385=1192.328,-45.371,-41.858,179.692,5.638,149.087
C04386=1192.333,-45.620,-41.846,179.689,5.637,149.088
C04387=1192.338,-45.870,-41.835,179.688,5.637,149.088
C04388=1192.343,-46.119,-41.822,179.685,5.637,149.089
C04389=1192.349,-46.369,-41.810,179.682,5.636,149.090
C04390=1192.354,-46.619,-41.799,179.680,5.637,149.090
C04391=1192.359,-46.869,-41.787,179.678,5.636,149.091
C04392=1192.364,-47.118,-41.774,179.675,5.635,149.092
C04393=1192.369,-47.368,-41.763,179.673,5.635,149.092
C04394=1192.375,-47.617,-41.751,179.671,5.635,149.093
C04395=1192.380,-47.867,-41.740,179.668,5.635,149.094
C04396=1192.385,-48.116,-41.727,179.666,5.634,149.094
C04397=1192.390,-48.366,-41.716,179.664,5.634,149.095
C04398=1192.395,-48.616,-41.704,179.661,5.634,149.096
C04399=1192.401,-48.866,-41.692,179.658,5.633,149.096
C04400=1192.406,-49.136,-41.679,179.656,5.633,149.097
C04401=1192.412,-49.406,-41.666,179.653,5.633,149.098
C04402=1192.417,-49.676,-41.653,179.651,5.633,149.098
C04403=1192.423,-49.947,-41.640,179.648,5.632,149.099
C04404=1192.428,-50.196,-41.629,179.646,5.632,149.100
C04405=1192.433,-50.446,-41.617,179.643,5.631,149.100
C04406=1192.439,-50.695,-41.606,179.641,5.632,149.101
C04407=1192.444,-50.945,-41.594,179.639,5.631,149.102
C04408=1192.449,-51.194,-41.582,179.636,5.630,149.102
C04409=1192.454,-51.444,-41.570,179.634,5.631,149.103
C04410=1192.459,-51.694,-41.559,179.632,5.630,149.104
C04411=1192.464,-51.944,-41.547,179.629,5.630,149.104
C04412=1192.470,-52.194,-41.535,179.627,5.629,149.105
C04413=1192.474,-52.443,-41.524,179.625,5.629,149.105
C04414=1192.480,-52.693,-41.512,179.622,5.629,149.106
C04415=1192.486,-52.943,-41.500,179.619,5.628,149.107
C04416=1192.491,-53.192,-41.489,179.617,5.629,149.108
C04417=1192.496,-53.442,-41.477,179.615,5.628,149.108
C04418=1192.501,-53.692,-41.466,179.612,5.628,149.109
C04419=1192.506,-53.941,-41.453,179.610,5.628,149.109
C04420=1192.510,-54.191,-41.442,179.608,5.627,149.110
C04421=1192.516,-54.441,-41.430,179.606,5.627,149.111
C04422=1192.521,-54.691,-41.418,179.603,5.627,149.111
C04423=1192.527,-54.939,-41.407,179.601,5.627,149.112
C04424=1192.532,-55.189,-41.395,179.598,5.626,149.113
C04425=1192.537,-55.439,-41.384,179.597,5.626,149.113
C04426=1192.542,-55.689,-41.372,179.594,5.626,149.114
C04427=1192.547,-55.939,-41.361,179.591,5.625,149.115
C04428=1192.552,-56.189,-41.349,179.589,5.625,149.115
C04429=1192.558,-56.437,-41.338,179.587,5.625,149.116
C04430=1192.563,-56.687,-41.326,179.584,5.624,149.117
C04431=1192.568,-56.937,-41.315,179.582,5.624,149.117
C04432=1192.573,-57.187,-41.303,179.580,5.624,149.118
C04433=1192.578,-57.437,-41.292,179.577,5.623,149.118
C04434=1192.583,-57.687,-41.280,179.575,5.623,149.119
C04435=1192.589,-57.935,-41.269,179.573,5.623,149.120
C04436=1192.594,-58.186,-41.258,179.570,5.623,149.121
C04437=1192.599,-58.436,-41.246,179.568,5.622,149.121
C04438=1192.604,-58.686,-41.234,179.566,5.623,149.122
C04439=1192.609,-58.935,-41.223,179.563,5.622,149.122
C04440=1192.615,-59.184,-41.212,179.560,5.622,149.123
C04441=1192.620,-59.434,-41.200,179.559,5.622,149.124
C04442=1192.625,-59.684,-41.188,179.556,5.621,149.124
C04443=1192.630,-59.934,-41.177,179.553,5.621,149.125
C04444=1192.636,-60.183,-41.166,179.551,5.621,149.126
C04445=1192.641,-60.432,-41.154,179.549,5.621,149.126
C04446=1192.646,-60.683,-41.144,179.546,5.620,149.127
C04447=1192.651,-60.933,-41.132,179.544,5.620,149.128
C04448=1192.656,-61.182,-41.121,179.542,5.620,149.128
C04449=1192.662,-61.431,-41.109,179.539,5.619,149.129
C04450=1192.667,-61.681,-41.098,179.537,5.619,149.129
C04451=1192.672,-61.931,-41.086,179.535,5.619,149.130
C04452=1192.677,-62.181,-41.075,179.532,5.618,149.131
C04453=1192.682,-62.430,-41.064,179.531,5.618,149.131
C04454=1192.688,-62.680,-41.053,179.528,5.618,149.132
C04455=1192.692,-62.930,-41.041,179.525,5.618,149.133
C04456=1192.698,-63.180,-41.029,179.523,5.618,149.133
C04457=1192.703,-63.429,-41.019,179.521,5.617,149.134
C04458=1192.708,-63.679,-41.008,179.518,5.617,149.135
C04459=1192.713,-63.929,-40.996,179.516,5.617,149.135
C04460=1192.719,-64.178,-40.985,179.513,5.617,149.136
C04461=1192.725,-64.428,-40.974,179.511,5.616,149.137
C04462=1192.729,-64.678,-40.963,179.509,5.616,149.137
C04463=1192.734,-64.928,-40.951,179.507,5.616,149.138
C04464=1192.740,-65.177,-40.940,179.504,5.616,149.139
C04465=1192.745,-65.427,-40.929,179.502,5.615,149.139
C04466=1192.750,-65.677,-40.918,179.500,5.615,149.140
C04467=1192.756,-65.926,-40.906,179.498,5.615,149.141
C04468=1192.760,-66.176,-40.895,179.495,5.615,149.141
C04469=1192.765,-66.426,-40.885,179.493,5.614,149.142
C04470=1192.771,-66.675,-40.873,179.491,5.614,149.142
C04471=1192.776,-66.925,-40.862,179.488,5.614,149.143
C04472=1192.781,-67.175,-40.851,179.485,5.614,149.144
C04473=1192.787,-67.424,-40.840,179.484,5.614,149.144
C04474=1192.792,-67.674,-40.828,179.481,5.613,149.145
C04475=1192.797,-67.924,-40.818,179.478,5.613,149.146
C04476=1192.802,-68.173,-40.807,179.476,5.613,149.146
C04477=1192.808,-68.423,-40.795,179.474,5.612,149.147
C04478=1192.813,-68.673,-40.784,179.472,5.613,149.148
C04479=1192.818,-68.922,-40.773,179.469,5.612,149.148
C04480=1192.824,-69.173,-40.762,179.467,5.612,149.149
C04481=1192.828,-69.422,-40.751,179.465,5.612,149.150
C04482=1192.834,-69.671,-40.740,179.462,5.611,149.150
C04483=1192.839,-69.921,-40.730,179.460,5.611,149.151
C04484=1192.844,-70.171,-40.718,179.458,5.611,149.151
C04485=1192.850,-70.421,-40.707,179.455,5.610,149.152
C04486=1192.854,-70.670,-40.696,179.453,5.610,149.153
C04487=1192.860,-70.920,-40.686,179.451,5.610,149.154
C04488=1192.865,-71.170,-40.674,179.449,5.610,149.154
C04489=1192.870,-71.420,-40.663,179.446,5.610,149.155
C04490=1192.876,-71.669,-40.653,179.444,5.610,149.155
C04491=1192.880,-71.919,-40.641,179.441,5.609,149.156
C04492=1192.886,-72.168,-40.631,179.439,5.609,149.157
C04493=1192.891,-72.418,-40.619,179.437,5.609,149.157
C04494=1192.896,-72.668,-40.609,179.434,5.608,149.158
C04495=1192.902,-72.917,-40.598,179.433,5.608,149.159
C04496=1192.907,-73.168,-40.587,179.430,5.608,149.159
C04497=1192.912,-73.417,-40.576,179.428,5.608,149.160
C04498=1192.918,-73.667,-40.565,179.425,5.608,149.161
C04499=1192.922,-73.917,-40.554,179.423,5.607,149.161
C04500=1192.928,-74.166,-40.543,179.421,5.607,149.162
C04501=1192.933,-74.416,-40.532,179.418,5.607,149.163
C04502=1192.938,-74.665,-40.522,179.416,5.607,149.163
C04503=1192.944,-74.915,-40.510,179.414,5.607,149.164
C04504=1192.949,-75.187,-40.499,179.411,5.606,149.164
C04505=1192.955,-75.457,-40.487,179.409,5.606,149.165
C04506=1192.961,-75.728,-40.475,179.406,5.606,149.166
C04507=1192.966,-75.999,-40.464,179.404,5.606,149.167
C04508=1192.971,-76.248,-40.453,179.401,5.605,149.167
C04509=1192.977,-76.499,-40.442,179.399,5.606,149.168
C04510=1192.982,-76.748,-40.431,179.397,5.605,149.168
C04511=1192.987,-76.998,-40.420,179.395,5.605,149.169
C04512=1192.993,-77.247,-40.410,179.392,5.605,149.170
C04513=1192.997,-77.497,-40.399,179.390,5.604,149.170
C04514=1193.003,-77.747,-40.389,179.388,5.604,149.171
C04515=1193.008,-77.997,-40.378,179.385,5.604,149.172
C04516=1193.013,-78.246,-40.367,179.383,5.603,149.173
C04517=1193.018,-78.496,-40.357,179.381,5.603,149.173
C04518=1193.024,-78.745,-40.346,179.378,5.603,149.174
C04519=1193.029,-78.995,-40.335,179.376,5.603,149.174
C04520=1193.035,-79.245,-40.324,179.374,5.603,149.175
C04521=1193.040,-79.495,-40.313,179.371,5.602,149.176
C04522=1193.045,-79.744,-40.303,179.369,5.603,149.176
C04523=1193.050,-79.994,-40.292,179.367,5.602,149.177
C04524=1193.056,-80.244,-40.282,179.365,5.602,149.177
C04525=1193.061,-80.494,-40.271,179.362,5.602,149.178
C04526=1193.066,-80.743,-40.261,179.360,5.601,149.179
C04527=1193.071,-80.993,-40.250,179.358,5.601,149.179
C04528=1193.076,-81.242,-40.239,179.355,5.601,149.180
C04529=1193.081,-81.493,-40.229,179.353,5.601,149.181
C04530=1193.087,-81.742,-40.218,179.351,5.600,149.181
C04531=1193.092,-81.992,-40.208,179.349,5.601,149.182
C04532=1193.097,-82.241,-40.197,179.346,5.600,149.183
C04533=1193.102,-82.492,-40.186,179.344,5.600,149.183
C04534=1193.108,-82.741,-40.176,179.342,5.600,149.184
C04535=1193.113,-82.991,-40.165,179.339,5.600,149.185
C04536=1193.118,-83.240,-40.155,179.337,5.600,149.185
C04537=1193.123,-83.490,-40.144,179.335,5.599,149.186
C04538=1193.129,-83.740,-40.134,179.332,5.599,149.187
C04539=1193.134,-83.990,-40.124,179.330,5.599,149.187
C04540=1193.139,-84.240,-40.113,179.328,5.598,149.188
C04541=1193.145,-84.489,-40.102,179.326,5.599,149.188
C04542=1193.150,-84.739,-40.092,179.323,5.598,149.189
C04543=1193.155,-84.989,-40.081,179.321,5.598,149.190
C04544=1193.160,-85.239,-40.071,179.319,5.598,149.190
C04545=1193.166,-85.488,-40.061,179.316,5.597,149.191
C04546=1193.170,-85.738,-40.051,179.314,5.598,149.192
C04547=1193.175,-85.987,-40.040,179.312,5.597,149.192
C04548=1193.181,-86.237,-40.029,179.310,5.597,149.193
C04549=1193.186,-86.487,-40.019,179.307,5.597,149.194
C04550=1193.192,-86.737,-40.009,179.305,5.596,149.194
C04551=1193.197,-86.987,-39.998,179.303,5.597,149.195
C04552=1193.202,-87.236,-39.988,179.300,5.596,149.196
C04553=1193.208,-87.486,-39.978,179.299,5.596,149.196
C04554=1193.213,-87.736,-39.967,179.296,5.596,149.197
C04555=1193.218,-87.985,-39.956,179.294,5.596,149.197
C04556=1193.223,-88.235,-39.946,179.291,5.596,149.198
C04557=1193.228,-88.484,-39.936,179.289,5.595,149.199
C04558=1193.234,-88.734,-39.926,179.287,5.595,149.199
C04559=1193.239,-88.984,-39.915,179.285,5.595,149.200
C04560=1193.244,-89.234,-39.905,179.283,5.595,149.201
C04561=1193.249,-89.484,-39.894,179.280,5.595,149.201
C04562=1193.255,-89.734,-39.884,179.278,5.595,149.202
C04563=1193.260,-89.983,-39.874,179.276,5.594,149.202
C04564=1193.265,-90.233,-39.864,179.273,5.594,149.203
C04565=1193.270,-90.483,-39.854,179.271,5.594,149.204
C04566=1193.276,-90.732,-39.844,179.269,5.593,149.204
C04567=1193.281,-90.982,-39.833,179.267,5.594,149.205
C04568=1193.286,-91.232,-39.823,179.264,5.593,149.206
C04569=1193.292,-91.481,-39.813,179.263,5.593,149.206
C04570=1193.296,-91.731,-39.803,179.260,5.593,149.207
C04571=1193.302,-91.981,-39.792,179.258,5.593,149.208
C04572=1193.307,-92.231,-39.782,179.256,5.592,149.208
C04573=1193.312,-92.481,-39.772,179.253,5.592,149.209
C04574=1193.318,-92.730,-39.761,179.251,5.592,149.210
C04575=1193.323,-92.980,-39.752,179.249,5.592,149.210
C04576=1193.328,-93.230,-39.741,179.247,5.592,149.211
C04577=1193.333,-93.479,-39.731,179.244,5.592,149.211
C04578=1193.339,-93.729,-39.721,179.242,5.592,149.212
C04579=1193.344,-93.979,-39.710,179.240,5.591,149.213
C04580=1193.349,-94.228,-39.701,179.238,5.592,149.213
C04581=1193.355,-94.478,-39.690,179.235,5.591,149.214
C04582=1193.360,-94.729,-39.681,179.233,5.590,149.215
C04583=1193.365,-94.978,-39.670,179.231,5.591,149.215
C04584=1193.370,-95.228,-39.661,179.229,5.590,149.216
C04585=1193.375,-95.478,-39.650,179.226,5.590,149.216
C04586=1193.381,-95.727,-39.640,179.224,5.590,149.217
C04587=1193.386,-95.977,-39.630,179.222,5.590,149.218
C04588=1193.391,-96.226,-39.620,179.219,5.590,149.218
C04589=1193.396,-96.476,-39.610,179.217,5.590,149.219
C04590=1193.402,-96.727,-39.600,179.215,5.589,149.220
C04591=1193.407,-96.976,-39.590,179.213,5.589,149.220
C04592=1193.413,-97.225,-39.580,179.210,5.589,149.221
C04593=1193.418,-97.476,-39.570,179.208,5.588,149.222
C04594=1193.423,-97.725,-39.559,179.206,5.589,149.222
C04595=1193.428,-97.974,-39.550,179.204,5.588,149.223
C04596=1193.434,-98.224,-39.540,179.202,5.588,149.223
C04597=1193.439,-98.475,-39.530,179.199,5.588,149.224
C04598=1193.444,-98.724,-39.520,179.197,5.588,149.225
C04599=1193.450,-98.973,-39.510,179.195,5.588,149.225
C04600=1193.455,-99.223,-39.500,179.193,5.588,149.226
C04601=1193.460,-99.474,-39.490,179.190,5.588,149.227
C04602=1193.465,-99.723,-39.480,179.189,5.588,149.227
C04603=1193.471,-99.973,-39.470,179.186,5.587,149.228
C04604=1193.476,-100.222,-39.460,179.183,5.587,149.229
C04605=1193.481,-100.473,-39.451,179.182,5.587,149.229
C04606=1193.487,-100.722,-39.440,179.179,5.586,149.230
C04607=1193.492,-100.972,-39.431,179.177,5.586,149.230
C04608=1193.498,-101.244,-39.420,179.175,5.586,149.231
C04609=1193.503,-101.515,-39.409,179.173,5.586,149.232
C04610=1193.509,-101.786,-39.398,179.170,5.586,149.232
C04611=1193.515,-102.058,-39.388,179.167,5.586,149.233
C04612=1193.520,-102.307,-39.378,179.165,5.586,149.234
C04613=1193.525,-102.558,-39.368,179.163,5.585,149.234
C04614=1193.530,-102.807,-39.358,179.161,5.586,149.235
C04615=1193.536,-103.057,-39.348,179.159,5.585,149.236
C04616=1193.541,-103.306,-39.338,179.157,5.585,149.236
C04617=1193.546,-103.556,-39.329,179.154,5.585,149.237
C04618=1193.551,-103.806,-39.319,179.152,5.585,149.237
C04619=1193.556,-104.056,-39.309,179.150,5.584,149.238
C04620=1193.562,-104.306,-39.299,179.147,5.584,149.239
C04621=1193.567,-104.555,-39.290,179.145,5.584,149.239
C04622=1193.573,-104.805,-39.280,179.143,5.584,149.240
C04623=1193.578,-105.055,-39.270,179.141,5.584,149.241
C04624=1193.583,-105.305,-39.260,179.138,5.583,149.241
C04625=1193.589,-105.555,-39.251,179.136,5.584,149.242
C04626=1193.593,-105.804,-39.241,179.134,5.583,149.243
C04627=1193.599,-106.054,-39.231,179.132,5.583,149.243
C04628=1193.604,-106.303,-39.222,179.129,5.583,149.244
C04629=1193.610,-106.553,-39.212,179.128,5.583,149.244
C04630=1193.614,-106.804,-39.203,179.125,5.582,149.245
C04631=1193.620,-107.053,-39.192,179.123,5.583,149.246
C04632=1193.625,-107.303,-39.183,179.121,5.582,149.246
C04633=1193.631,-107.552,-39.173,179.119,5.582,149.247
C04634=1193.636,-107.802,-39.164,179.117,5.582,149.248
C04635=1193.642,-108.052,-39.154,179.114,5.582,149.248
C04636=1193.646,-108.301,-39.144,179.112,5.582,149.249
C04637=1193.652,-108.551,-39.135,179.110,5.582,149.249
C04638=1193.657,-108.801,-39.125,179.108,5.581,149.250
C04639=1193.662,-109.051,-39.116,179.106,5.581,149.251
C04640=1193.667,-109.301,-39.106,179.103,5.581,149.251
C04641=1193.673,-109.551,-39.096,179.101,5.581,149.252
C04642=1193.678,-109.800,-39.087,179.099,5.580,149.253
C04643=1193.684,-110.050,-39.077,179.097,5.581,149.253
C04644=1193.689,-110.299,-39.068,179.094,5.580,149.254
C04645=1193.695,-110.550,-39.058,179.093,5.580,149.254
C04646=1193.700,-110.799,-39.049,179.090,5.580,149.255
C04647=1193.705,-111.050,-39.039,179.088,5.580,149.256
C04648=1193.710,-111.299,-39.029,179.086,5.580,149.256
C04649=1193.715,-111.549,-39.020,179.084,5.580,149.257
C04650=1193.721,-111.798,-39.010,179.081,5.579,149.258
C04651=1193.726,-112.048,-39.001,179.079,5.580,149.258
C04652=1193.732,-112.298,-38.992,179.077,5.579,149.259
C04653=1193.736,-112.548,-38.982,179.075,5.579,149.260
C04654=1193.742,-112.797,-38.973,179.072,5.579,149.260
C04655=1193.747,-113.047,-38.963,179.071,5.579,149.261
C04656=1193.752,-113.297,-38.954,179.068,5.578,149.261
C04657=1193.758,-113.546,-38.944,179.066,5.578,149.262
C04658=1193.763,-113.796,-38.935,179.064,5.578,149.263
C04659=1193.768,-114.046,-38.926,179.062,5.578,149.263
C04660=1193.774,-114.296,-38.916,179.060,5.578,149.264
C04661=1193.779,-114.545,-38.907,179.057,5.578,149.265
C04662=1193.785,-114.796,-38.897,179.055,5.577,149.265
C04663=1193.790,-115.045,-38.888,179.053,5.578,149.266
C04664=1193.794,-115.295,-38.879,179.051,5.577,149.266
C04665=1193.800,-115.545,-38.868,179.049,5.577,149.267
C04666=1193.805,-115.795,-38.859,179.046,5.577,149.268
C04667=1193.810,-116.045,-38.851,179.045,5.577,149.268
C04668=1193.816,-116.294,-38.840,179.042,5.577,149.269
C04669=1193.821,-116.544,-38.831,179.040,5.577,149.269
C04670=1193.826,-116.794,-38.822,179.038,5.576,149.270
C04671=1193.832,-117.043,-38.812,179.036,5.577,149.271
C04672=1193.837,-117.293,-38.803,179.033,5.576,149.271
C04673=1193.842,-117.543,-38.794,179.031,5.576,149.272
C04674=1193.848,-117.793,-38.785,179.029,5.575,149.272
C04675=1193.853,-118.042,-38.775,179.027,5.576,149.273
C04676=1193.858,-118.292,-38.766,179.025,5.575,149.274
C04677=1193.864,-118.543,-38.757,179.023,5.575,149.274
C04678=1193.869,-118.792,-38.747,179.020,5.575,149.275
C04679=1193.874,-119.042,-38.738,179.018,5.575,149.276
C04680=1193.880,-119.292,-38.729,179.016,5.575,149.276
C04681=1193.885,-119.542,-38.720,179.014,5.575,149.277
C04682=1193.890,-119.791,-38.710,179.011,5.574,149.278
C04683=1193.895,-120.041,-38.702,179.010,5.574,149.278
C04684=1193.901,-120.291,-38.692,179.007,5.574,149.279
C04685=1193.906,-120.541,-38.683,179.006,5.574,149.279
C04686=1193.911,-120.791,-38.674,179.003,5.574,149.280
C04687=1193.917,-121.039,-38.665,179.001,5.574,149.281
C04688=1193.923,-121.289,-38.656,178.999,5.573,149.281
C04689=1193.928,-121.539,-38.647,178.997,5.574,149.282
C04690=1193.933,-121.789,-38.638,178.994,5.573,149.282
C04691=1193.938,-122.039,-38.629,178.992,5.573,149.283
C04692=1193.944,-122.288,-38.619,178.990,5.572,149.284
C04693=1193.949,-122.538,-38.610,178.988,5.573,149.284
C04694=1193.954,-122.788,-38.601,178.986,5.573,149.285
C04695=1193.959,-123.038,-38.592,178.984,5.572,149.285
C04696=1193.965,-123.288,-38.583,178.982,5.573,149.286
C04697=1193.970,-123.538,-38.574,178.979,5.572,149.287
C04698=1193.975,-123.787,-38.564,178.977,5.572,149.287
C04699=1193.980,-124.037,-38.555,178.975,5.572,149.288
C04700=1193.986,-124.287,-38.546,178.973,5.572,149.289
C04701=1193.991,-124.537,-38.537,178.971,5.571,149.289
C04702=1193.997,-124.787,-38.528,178.969,5.572,149.290
C04703=1194.002,-125.036,-38.519,178.967,5.571,149.290
C04704=1194.008,-125.286,-38.510,178.965,5.571,149.291
C04705=1194.013,-125.536,-38.501,178.962,5.571,149.291
C04706=1194.018,-125.786,-38.493,178.960,5.571,149.292
C04707=1194.024,-126.035,-38.482,178.958,5.571,149.293
C04708=1194.029,-126.285,-38.473,178.956,5.571,149.293
C04709=1194.034,-126.535,-38.465,178.953,5.570,149.294
C04710=1194.039,-126.785,-38.456,178.952,5.570,149.295
C04711=1194.044,-127.035,-38.447,178.950,5.571,149.295
C04712=1193.623,-127.045,-38.485,178.946,5.574,149.297
C04713=1193.618,-126.796,-38.494,178.948,5.573,149.296
C04714=1193.613,-126.546,-38.503,178.950,5.574,149.296
C04715=1193.607,-126.296,-38.513,178.952,5.574,149.295
C04716=1193.602,-126.046,-38.522,178.954,5.575,149.295
C04717=1193.597,-125.797,-38.531,178.956,5.574,149.294
C04718=1193.592,-125.547,-38.540,178.958,5.574,149.294
C04719=1193.586,-125.297,-38.549,178.961,5.575,149.293
C04720=1193.581,-125.047,-38.558,178.962,5.575,149.292
C04721=1193.575,-124.798,-38.567,178.965,5.575,149.292
C04722=1193.570,-124.548,-38.576,178.966,5.575,149.291
C04723=1193.564,-124.298,-38.585,178.969,5.575,149.290
C04724=1193.559,-124.048,-38.594,178.971,5.575,149.290
C04725=1193.554,-123.798,-38.603,178.973,5.576,149.289
C04726=1193.549,-123.549,-38.612,178.976,5.575,149.288
C04727=1193.543,-123.299,-38.622,178.978,5.576,149.288
C04728=1193.538,-123.049,-38.631,178.980,5.576,149.287
C04729=1193.533,-122.799,-38.640,178.982,5.576,149.287
C04730=1193.528,-122.549,-38.649,178.984,5.576,149.286
C04731=1193.522,-122.299,-38.658,178.986,5.577,149.286
C04732=1193.517,-122.050,-38.668,178.988,5.576,149.285
C04733=1193.512,-121.800,-38.677,178.991,5.577,149.284
C04734=1193.507,-121.550,-38.685,178.993,5.577,149.284
C04735=1193.502,-121.300,-38.694,178.995,5.577,149.283
C04736=1193.496,-121.050,-38.704,178.997,5.577,149.282
C04737=1193.490,-120.801,-38.712,178.999,5.577,149.282
C04738=1193.485,-120.552,-38.722,179.001,5.578,149.281
C04739=1193.480,-120.302,-38.731,179.003,5.577,149.281
C04740=1193.474,-120.052,-38.740,179.005,5.578,149.280
C04741=1193.469,-119.802,-38.749,179.008,5.577,149.279
C04742=1193.464,-119.553,-38.759,179.010,5.578,149.279
C04743=1193.458,-119.302,-38.768,179.012,5.578,149.278
C04744=1193.453,-119.053,-38.777,179.015,5.578,149.277
C04745=1193.448,-118.803,-38.786,179.016,5.578,149.277
C04746=1193.443,-118.553,-38.796,179.019,5.579,149.276
C04747=1193.437,-118.303,-38.805,179.020,5.579,149.276
C04748=1193.432,-118.053,-38.814,179.023,5.579,149.275
C04749=1193.427,-117.804,-38.823,179.025,5.579,149.275
C04750=1193.421,-117.554,-38.833,179.027,5.579,149.274
C04751=1193.416,-117.304,-38.842,179.029,5.579,149.273
C04752=1193.411,-117.054,-38.851,179.032,5.580,149.273
C04753=1193.405,-116.805,-38.861,179.034,5.579,149.272
C04754=1193.400,-116.555,-38.870,179.036,5.580,149.271
C04755=1193.395,-116.305,-38.879,179.038,5.580,149.271
C04756=1193.389,-116.056,-38.889,179.040,5.581,149.270
C04757=1193.384,-115.806,-38.898,179.042,5.580,149.270
C04758=1193.379,-115.556,-38.907,179.045,5.581,149.269
C04759=1193.373,-115.306,-38.917,179.047,5.581,149.268
C04760=1193.368,-115.056,-38.926,179.049,5.581,149.268
C04761=1193.363,-114.807,-38.935,179.051,5.581,149.267
C04762=1193.358,-114.556,-38.946,179.054,5.581,149.266
C04763=1193.353,-114.307,-38.955,179.056,5.581,149.266
C04764=1193.347,-114.057,-38.963,179.058,5.582,149.265
C04765=1193.342,-113.807,-38.974,179.060,5.581,149.264
C04766=1193.337,-113.557,-38.983,179.062,5.582,149.264
C04767=1193.331,-113.308,-38.993,179.064,5.582,149.263
C04768=1193.326,-113.058,-39.002,179.066,5.582,149.263
C04769=1193.321,-112.808,-39.011,179.068,5.582,149.262
C04770=1193.315,-112.558,-39.021,179.071,5.582,149.261
C04771=1193.310,-112.309,-39.030,179.073,5.582,149.261
C04772=1193.304,-112.059,-39.040,179.075,5.583,149.260
C04773=1193.299,-111.809,-39.049,179.077,5.583,149.260
C04774=1193.294,-111.560,-39.059,179.080,5.583,149.259
C04775=1193.289,-111.310,-39.068,179.082,5.583,149.258
C04776=1193.283,-111.060,-39.077,179.084,5.584,149.258
C04777=1193.278,-110.810,-39.087,179.086,5.583,149.257
C04778=1193.273,-110.560,-39.096,179.088,5.584,149.257
C04779=1193.268,-110.310,-39.106,179.090,5.584,149.256
C04780=1193.262,-110.061,-39.115,179.093,5.584,149.255
C04781=1193.257,-109.811,-39.126,179.095,5.584,149.255
C04782=1193.252,-109.561,-39.134,179.097,5.584,149.254
C04783=1193.246,-109.312,-39.145,179.099,5.584,149.253
C04784=1193.241,-109.062,-39.154,179.102,5.585,149.253
C04785=1193.235,-108.812,-39.164,179.104,5.584,149.252
C04786=1193.230,-108.562,-39.173,179.106,5.585,149.252
C04787=1193.225,-108.312,-39.183,179.108,5.585,149.251
C04788=1193.220,-108.063,-39.193,179.111,5.585,149.250
C04789=1193.214,-107.813,-39.202,179.112,5.585,149.250
C04790=1193.209,-107.563,-39.212,179.115,5.586,149.249
C04791=1193.204,-107.313,-39.221,179.116,5.586,149.248
C04792=1193.199,-107.064,-39.231,179.119,5.586,149.248
C04793=1193.193,-106.814,-39.241,179.121,5.586,149.247
C04794=1193.188,-106.565,-39.250,179.123,5.586,149.247
C04795=1193.183,-106.314,-39.260,179.125,5.586,149.246
C04796=1193.178,-106.065,-39.270,179.128,5.587,149.245
C04797=1193.172,-105.815,-39.280,179.130,5.586,149.245
C04798=1193.167,-105.565,-39.289,179.132,5.587,149.244
C04799=1193.161,-105.316,-39.299,179.135,5.587,149.243
C04800=1193.156,-105.066,-39.308,179.137,5.587,149.243
C04801=1193.151,-104.816,-39.318,179.139,5.587,149.242
C04802=1193.146,-104.566,-39.328,179.141,5.587,149.242
C04803=1193.141,-104.316,-39.338,179.144,5.588,149.241
C04804=1193.135,-104.067,-39.348,179.145,5.588,149.240
C04805=1193.130,-103.817,-39.357,179.148,5.588,149.240
C04806=1193.124,-103.567,-39.367,179.150,5.588,149.239
C04807=1193.120,-103.317,-39.377,179.152,5.589,149.238
C04808=1193.114,-103.068,-39.387,179.154,5.588,149.238
C04809=1193.109,-102.818,-39.396,179.157,5.589,149.237
C04810=1193.104,-102.568,-39.406,179.159,5.589,149.236
C04811=1193.098,-102.319,-39.416,179.161,5.589,149.236
C04812=1193.093,-102.068,-39.426,179.163,5.589,149.235
C04813=1193.087,-101.797,-39.437,179.166,5.589,149.235
C04814=1193.081,-101.525,-39.447,179.168,5.590,149.234
C04815=1193.076,-101.254,-39.458,179.170,5.589,149.233
C04816=1193.070,-100.982,-39.469,179.173,5.590,149.232
C04817=1193.065,-100.733,-39.478,179.176,5.590,149.232
C04818=1193.059,-100.483,-39.489,179.177,5.590,149.231
C04819=1193.055,-100.234,-39.498,179.180,5.591,149.231
C04820=1193.050,-99.984,-39.509,179.182,5.590,149.230
C04821=1193.044,-99.733,-39.518,179.184,5.591,149.229
C04822=1193.039,-99.484,-39.528,179.186,5.591,149.229
C04823=1193.033,-99.235,-39.538,179.188,5.591,149.228
C04824=1193.028,-98.984,-39.549,179.191,5.591,149.227
C04825=1193.023,-98.735,-39.558,179.193,5.591,149.227
C04826=1193.017,-98.485,-39.568,179.195,5.591,149.226
C04827=1193.012,-98.236,-39.578,179.198,5.592,149.226
C04828=1193.007,-97.986,-39.588,179.200,5.591,149.225
C04829=1193.002,-97.736,-39.598,179.202,5.592,149.224
C04830=1192.996,-97.486,-39.608,179.204,5.593,149.224
C04831=1192.991,-97.236,-39.618,179.207,5.592,149.223
C04832=1192.986,-96.986,-39.628,179.209,5.593,149.222
C04833=1192.981,-96.737,-39.638,179.211,5.593,149.222
C04834=1192.975,-96.487,-39.648,179.213,5.593,149.221
C04835=1192.970,-96.238,-39.658,179.215,5.593,149.220
C04836=1192.965,-95.987,-39.668,179.218,5.594,149.220
C04837=1192.959,-95.738,-39.678,179.220,5.593,149.219
C04838=1192.954,-95.488,-39.688,179.222,5.594,149.219
C04839=1192.949,-95.239,-39.698,179.224,5.594,149.218
C04840=1192.944,-94.989,-39.708,179.227,5.594,149.217
C04841=1192.938,-94.739,-39.719,179.229,5.595,149.217
C04842=1192.933,-94.490,-39.729,179.231,5.594,149.216
C04843=1192.928,-94.240,-39.739,179.234,5.595,149.215
C04844=1192.923,-93.990,-39.749,179.235,5.595,149.215
C04845=1192.917,-93.741,-39.759,179.238,5.595,149.214
C04846=1192.912,-93.490,-39.769,179.240,5.595,149.213
C04847=1192.907,-93.240,-39.779,179.242,5.596,149.213
C04848=1192.901,-92.991,-39.789,179.244,5.595,149.212
C04849=1192.896,-92.741,-39.799,179.247,5.596,149.211
C04850=1192.891,-92.491,-39.810,179.249,5.596,149.211
C04851=1192.885,-92.242,-39.820,179.251,5.596,149.210
C04852=1192.881,-91.992,-39.830,179.254,5.596,149.210
C04853=1192.875,-91.742,-39.840,179.256,5.596,149.209
C04854=1192.870,-91.493,-39.850,179.258,5.597,149.208
C04855=1192.865,-91.242,-39.861,179.260,5.596,149.208
C04856=1192.859,-90.993,-39.871,179.263,5.597,149.207
C04857=1192.854,-90.743,-39.881,179.265,5.598,149.206
C04858=1192.849,-90.493,-39.891,179.267,5.597,149.206
C04859=1192.844,-90.244,-39.901,179.269,5.598,149.205
C04860=1192.838,-89.994,-39.912,179.272,5.598,149.205
C04861=1192.833,-89.744,-39.922,179.274,5.598,149.204
C04862=1192.828,-89.494,-39.932,179.276,5.598,149.203
C04863=1192.822,-89.245,-39.943,179.279,5.598,149.203
C04864=1192.818,-88.995,-39.953,179.281,5.598,149.202
C04865=1192.812,-88.745,-39.963,179.283,5.599,149.201
C04866=1192.807,-88.495,-39.973,179.285,5.599,149.201
C04867=1192.802,-88.246,-39.984,179.288,5.599,149.200
C04868=1192.796,-87.997,-39.995,179.290,5.600,149.200
C04869=1192.791,-87.746,-40.005,179.292,5.599,149.199
C04870=1192.786,-87.497,-40.015,179.294,5.600,149.198
C04871=1192.781,-87.247,-40.026,179.296,5.600,149.198
C04872=1192.775,-86.997,-40.036,179.299,5.600,149.197
C04873=1192.770,-86.748,-40.046,179.301,5.601,149.196
C04874=1192.765,-86.498,-40.056,179.303,5.601,149.196
C04875=1192.760,-86.248,-40.066,179.306,5.601,149.195
C04876=1192.755,-85.998,-40.077,179.308,5.601,149.194
C04877=1192.749,-85.749,-40.088,179.310,5.601,149.194
C04878=1192.744,-85.499,-40.098,179.313,5.602,149.193
C04879=1192.739,-85.249,-40.109,179.315,5.601,149.192
C04880=1192.733,-85.000,-40.119,179.317,5.602,149.192
C04881=1192.728,-84.749,-40.130,179.319,5.602,149.191
C04882=1192.722,-84.500,-40.140,179.322,5.602,149.191
C04883=1192.718,-84.250,-40.151,179.324,5.602,149.190
C04884=1192.712,-84.001,-40.161,179.326,5.603,149.189
C04885=1192.707,-83.750,-40.172,179.329,5.603,149.189
C04886=1192.702,-83.501,-40.182,179.331,5.603,149.188
C04887=1192.696,-83.251,-40.192,179.333,5.604,149.187
C04888=1192.691,-83.002,-40.204,179.335,5.603,149.187
C04889=1192.686,-82.752,-40.213,179.338,5.604,149.186
C04890=1192.681,-82.502,-40.224,179.340,5.604,149.185
C04891=1192.676,-82.253,-40.234,179.342,5.604,149.185
C04892=1192.671,-82.003,-40.245,179.345,5.604,149.184
C04893=1192.666,-81.753,-40.255,179.347,5.604,149.183
C04894=1192.660,-81.503,-40.267,179.349,5.605,149.183
C04895=1192.654,-81.253,-40.277,179.352,5.605,149.182
C04896=1192.650,-81.004,-40.288,179.354,5.605,149.181
C04897=1192.644,-80.754,-40.298,179.356,5.606,149.181
C04898=1192.639,-80.504,-40.309,179.358,5.605,149.180
C04899=1192.633,-80.254,-40.319,179.361,5.606,149.180
C04900=1192.629,-80.005,-40.330,179.363,5.606,149.179
C04901=1192.623,-79.755,-40.341,179.365,5.606,149.178
C04902=1192.618,-79.505,-40.351,179.367,5.607,149.178
C04903=1192.613,-79.256,-40.362,179.370,5.606,149.177
C04904=1192.608,-79.006,-40.373,179.372,5.607,149.176
C04905=1192.602,-78.756,-40.383,179.374,5.607,149.176
C04906=1192.597,-78.507,-40.394,179.377,5.607,149.175
C04907=1192.592,-78.257,-40.404,179.379,5.607,149.174
C04908=1192.587,-78.007,-40.415,179.381,5.607,149.174
C04909=1192.582,-77.758,-40.426,179.383,5.608,149.173
C04910=1192.577,-77.508,-40.436,179.386,5.608,149.172
C04911=1192.571,-77.258,-40.448,179.388,5.608,149.172
C04912=1192.566,-77.008,-40.459,179.390,5.609,149.171
C04913=1192.560,-76.759,-40.469,179.392,5.608,149.171
C04914=1192.555,-76.509,-40.480,179.395,5.609,149.170
C04915=1192.550,-76.260,-40.490,179.397,5.610,149.169
C04916=1192.545,-76.009,-40.501,179.399,5.609,149.169
C04917=1192.539,-75.738,-40.513,179.402,5.610,149.168
C04918=1192.534,-75.468,-40.524,179.405,5.610,149.167
C04919=1192.528,-75.197,-40.537,179.407,5.610,149.167
C04920=1192.522,-74.926,-40.548,179.410,5.610,149.166
C04921=1192.517,-74.677,-40.559,179.412,5.611,149.165
C04922=1192.512,-74.427,-40.570,179.414,5.610,149.165
C04923=1192.506,-74.178,-40.581,179.416,5.611,149.164
C04924=1192.501,-73.927,-40.592,179.419,5.611,149.163
C04925=1192.495,-73.678,-40.603,179.421,5.611,149.163
C04926=1192.490,-73.428,-40.613,179.423,5.612,149.162
C04927=1192.486,-73.178,-40.625,179.426,5.612,149.161
C04928=1192.480,-72.929,-40.635,179.428,5.612,149.161
C04929=1192.475,-72.679,-40.646,179.430,5.613,149.160
C04930=1192.469,-72.429,-40.657,179.432,5.612,149.159
C04931=1192.464,-72.180,-40.668,179.435,5.613,149.159
C04932=1192.459,-71.929,-40.679,179.437,5.613,149.158
C04933=1192.454,-71.680,-40.690,179.439,5.613,149.158
C04934=1192.448,-71.430,-40.701,179.442,5.614,149.157
C04935=1192.443,-71.181,-40.712,179.445,5.614,149.156
C04936=1192.438,-70.931,-40.722,179.446,5.614,149.156
C04937=1192.433,-70.681,-40.734,179.449,5.614,149.155
C04938=1192.428,-70.432,-40.744,179.451,5.614,149.154
C04939=1192.422,-70.182,-40.756,179.454,5.614,149.154
C04940=1192.417,-69.933,-40.767,179.456,5.615,149.153
C04941=1192.412,-69.682,-40.777,179.458,5.615,149.152
C04942=1192.407,-69.433,-40.788,179.461,5.615,149.152
C04943=1192.401,-69.183,-40.799,179.463,5.616,149.151
C04944=1192.396,-68.933,-40.811,179.465,5.616,149.150
C04945=1192.392,-68.684,-40.822,179.468,5.616,149.150
C04946=1192.385,-68.434,-40.833,179.470,5.616,149.149
C04947=1192.381,-68.184,-40.844,179.472,5.617,149.149
C04948=1192.376,-67.934,-40.855,179.475,5.617,149.148
C04949=1192.370,-67.685,-40.865,179.477,5.617,149.147
C04950=1192.365,-67.435,-40.877,179.479,5.617,149.146
C04951=1192.360,-67.185,-40.888,179.481,5.618,149.146
C04952=1192.355,-66.936,-40.899,179.484,5.618,149.145
C04953=1192.349,-66.686,-40.911,179.486,5.618,149.145
C04954=1192.344,-66.436,-40.921,179.489,5.618,149.144
C04955=1192.339,-66.187,-40.932,179.490,5.618,149.143
C04956=1192.333,-65.937,-40.944,179.493,5.619,149.143
C04957=1192.328,-65.687,-40.955,179.496,5.619,149.142
C04958=1192.323,-65.438,-40.966,179.497,5.619,149.141
C04959=1192.318,-65.188,-40.977,179.500,5.620,149.141
C04960=1192.313,-64.938,-40.989,179.502,5.619,149.140
C04961=1192.307,-64.689,-40.999,179.505,5.620,149.139
C04962=1192.302,-64.439,-41.011,179.507,5.621,149.139
C04963=1192.297,-64.189,-41.022,179.509,5.620,149.138
C04964=1192.293,-63.939,-41.033,179.512,5.621,149.137
C04965=1192.286,-63.690,-41.044,179.514,5.621,149.137
C04966=1192.282,-63.440,-41.056,179.516,5.621,149.136
C04967=1192.276,-63.190,-41.067,179.519,5.621,149.136
C04968=1192.271,-62.940,-41.079,179.521,5.622,149.135
C04969=1192.266,-62.691,-41.089,179.523,5.622,149.134
C04970=1192.260,-62.441,-41.101,179.526,5.622,149.134
C04971=1192.256,-62.191,-41.112,179.528,5.623,149.133
C04972=1192.250,-61.942,-41.124,179.530,5.622,149.132
C04973=1192.245,-61.692,-41.135,179.533,5.623,149.132
C04974=1192.240,-61.443,-41.146,179.535,5.624,149.131
C04975=1192.235,-61.192,-41.157,179.537,5.623,149.130
C04976=1192.230,-60.943,-41.169,179.540,5.624,149.130
C04977=1192.224,-60.693,-41.180,179.543,5.624,149.129
C04978=1192.219,-60.444,-41.191,179.544,5.624,149.129
C04979=1192.214,-60.194,-41.203,179.547,5.625,149.128
C04980=1192.209,-59.944,-41.215,179.550,5.625,149.127
C04981=1192.204,-59.695,-41.226,179.552,5.625,149.126
C04982=1192.198,-59.445,-41.237,179.554,5.625,149.126
C04983=1192.193,-59.195,-41.248,179.556,5.626,149.125
C04984=1192.188,-58.945,-41.260,179.559,5.626,149.125
C04985=1192.183,-58.696,-41.271,179.561,5.626,149.124
C04986=1192.177,-58.446,-41.283,179.563,5.627,149.123
C04987=1192.173,-58.197,-41.294,179.565,5.626,149.123
C04988=1192.167,-57.947,-41.306,179.568,5.627,149.122
C04989=1192.162,-57.697,-41.317,179.571,5.627,149.121
C04990=1192.157,-57.447,-41.329,179.572,5.627,149.121
C04991=1192.152,-57.198,-41.340,179.575,5.628,149.120
C04992=1192.146,-56.948,-41.352,179.578,5.628,149.119
C04993=1192.142,-56.699,-41.363,179.580,5.628,149.119
C04994=1192.136,-56.449,-41.375,179.582,5.629,149.118
C04995=1192.131,-56.199,-41.386,179.585,5.629,149.117
C04996=1192.125,-55.950,-41.398,179.587,5.629,149.117
C04997=1192.121,-55.700,-41.409,179.589,5.629,149.116
C04998=1192.115,-55.450,-41.421,179.592,5.630,149.116
C04999=1192.111,-55.201,-41.432,179.594,5.630,149.115
C05000=1192.105,-54.951,-41.444,179.596,5.630,149.114
C05001=1192.100,-54.701,-41.455,179.599,5.630,149.113
C05002=1192.095,-54.451,-41.467,179.601,5.631,149.113
C05003=1192.089,-54.202,-41.479,179.603,5.631,149.112
C05004=1192.084,-53.952,-41.490,179.606,5.631,149.112
C05005=1192.079,-53.702,-41.502,179.609,5.632,149.111
C05006=1192.074,-53.453,-41.513,179.610,5.632,149.110
C05007=1192.069,-53.203,-41.525,179.613,5.632,149.110
C05008=1192.064,-52.953,-41.537,179.616,5.633,149.109
C05009=1192.059,-52.703,-41.548,179.618,5.632,149.108
C05010=1192.053,-52.453,-41.560,179.620,5.633,149.108
C05011=1192.048,-52.204,-41.571,179.622,5.634,149.107
C05012=1192.043,-51.955,-41.583,179.625,5.634,149.106
C05013=1192.037,-51.705,-41.595,179.627,5.634,149.106
C05014=1192.033,-51.456,-41.607,179.630,5.634,149.105
C05015=1192.027,-51.206,-41.619,179.632,5.635,149.105
C05016=1192.023,-50.956,-41.630,179.634,5.635,149.104
C05017=1192.017,-50.706,-41.642,179.637,5.635,149.103
C05018=1192.012,-50.456,-41.654,179.639,5.635,149.102
C05019=1192.007,-50.207,-41.665,179.641,5.636,149.102
C05020=1192.001,-49.957,-41.677,179.644,5.636,149.101
C05021=1191.996,-49.687,-41.690,179.646,5.636,149.101
C05022=1191.990,-49.417,-41.703,179.649,5.637,149.100
C05023=1191.984,-49.147,-41.715,179.652,5.637,149.099
C05024=1191.979,-48.877,-41.728,179.654,5.638,149.098
C05025=1191.974,-48.627,-41.740,179.656,5.637,149.098
C05026=1191.968,-48.377,-41.752,179.659,5.638,149.097
C05027=1191.964,-48.128,-41.764,179.661,5.639,149.097
C05028=1191.958,-47.878,-41.776,179.663,5.638,149.096
C05029=1191.953,-47.628,-41.788,179.666,5.639,149.095
C05030=1191.948,-47.378,-41.799,179.669,5.639,149.094
C05031=1191.943,-47.128,-41.811,179.671,5.640,149.094
C05032=1191.937,-46.880,-41.823,179.673,5.640,149.093
C05033=1191.932,-46.630,-41.835,179.676,5.640,149.093
C05034=1191.927,-46.380,-41.846,179.678,5.640,149.092
C05035=1191.922,-46.130,-41.858,179.680,5.641,149.091
C05036=1191.917,-45.881,-41.871,179.683,5.641,149.091
C05037=1191.911,-45.631,-41.883,179.685,5.641,149.090
C05038=1191.906,-45.381,-41.894,179.688,5.642,149.089
C05039=1191.901,-45.132,-41.907,179.690,5.641,149.089
C05040=1191.896,-44.882,-41.919,179.692,5.642,149.088
C05041=1191.890,-44.632,-41.930,179.695,5.643,149.087
C05042=1191.886,-44.383,-41.942,179.698,5.643,149.087
C05043=1191.881,-44.133,-41.954,179.700,5.643,149.086
C05044=1191.875,-43.883,-41.966,179.702,5.644,149.086
C05045=1191.870,-43.634,-41.979,179.704,5.644,149.085
C05046=1191.865,-43.384,-41.991,179.707,5.644,149.084
C05047=1191.860,-43.134,-42.002,179.709,5.644,149.083
C05048=1191.855,-42.885,-42.015,179.711,5.645,149.083
C05049=1191.849,-42.635,-42.026,179.714,5.645,149.082
C05050=1191.844,-42.385,-42.038,179.716,5.645,149.082
C05051=1191.839,-42.136,-42.051,179.719,5.646,149.081
C05052=1191.833,-41.886,-42.063,179.721,5.646,149.080
C05053=1191.829,-41.637,-42.075,179.724,5.647,149.080
C05054=1191.824,-41.387,-42.087,179.726,5.647,149.079
C05055=1191.818,-41.138,-42.099,179.728,5.647,149.078
C05056=1191.813,-40.888,-42.111,179.731,5.647,149.078
C05057=1191.808,-40.637,-42.123,179.733,5.648,149.077
C05058=1191.803,-40.388,-42.136,179.735,5.648,149.076
C05059=1191.798,-40.138,-42.148,179.738,5.648,149.076
C05060=1191.793,-39.889,-42.160,179.741,5.649,149.075
C05061=1191.788,-39.639,-42.172,179.743,5.650,149.075
C05062=1191.783,-39.390,-42.184,179.745,5.649,149.074
C05063=1191.777,-39.140,-42.196,179.748,5.650,149.073
C05064=1191.772,-38.890,-42.209,179.750,5.650,149.072
C05065=1191.767,-38.640,-42.221,179.753,5.651,149.072
C05066=1191.762,-38.391,-42.233,179.754,5.651,149.071
C05067=1191.756,-38.141,-42.245,179.757,5.651,149.071
C05068=1191.751,-37.892,-42.258,179.760,5.652,149.070
C05069=1191.746,-37.642,-42.270,179.762,5.652,149.069
C05070=1191.740,-37.393,-42.282,179.764,5.652,149.069
C05071=1191.736,-37.143,-42.294,179.767,5.652,149.068
C05072=1191.731,-36.893,-42.307,179.769,5.653,149.067
C05073=1191.726,-36.643,-42.319,179.772,5.653,149.067
C05074=1191.721,-36.394,-42.331,179.774,5.653,149.066
C05075=1191.716,-36.144,-42.344,179.776,5.654,149.065
C05076=1191.710,-35.894,-42.356,179.779,5.654,149.065
C05077=1191.705,-35.645,-42.368,179.782,5.655,149.064
C05078=1191.700,-35.395,-42.380,179.784,5.654,149.063
C05079=1191.694,-35.146,-42.393,179.786,5.655,149.063
C05080=1191.689,-34.896,-42.405,179.789,5.656,149.062
C05081=1191.685,-34.646,-42.418,179.791,5.656,149.061
C05082=1191.679,-34.397,-42.430,179.793,5.656,149.061
C05083=1191.674,-34.147,-42.442,179.796,5.656,149.060
C05084=1191.669,-33.897,-42.455,179.798,5.657,149.060
C05085=1191.664,-33.648,-42.467,179.801,5.658,149.059
C05086=1191.658,-33.398,-42.479,179.803,5.658,149.058
C05087=1191.653,-33.149,-42.492,179.805,5.658,149.057
C05088=1191.649,-32.899,-42.505,179.808,5.658,149.057
C05089=1191.643,-32.649,-42.517,179.810,5.659,149.056
C05090=1191.638,-32.399,-42.529,179.813,5.659,149.056
C05091=1191.633,-32.150,-42.542,179.815,5.659,149.055
C05092=1191.628,-31.900,-42.554,179.818,5.659,149.054
C05093=1191.622,-31.651,-42.566,179.820,5.660,149.054
C05094=1191.618,-31.401,-42.579,179.823,5.661,149.053
C05095=1191.612,-31.151,-42.592,179.825,5.661,149.052
C05096=1191.607,-30.901,-42.604,179.827,5.661,149.052
C05097=1191.601,-30.652,-42.617,179.829,5.662,149.051
C05098=1191.596,-30.403,-42.630,179.832,5.662,149.050
C05099=1191.591,-30.153,-42.642,179.835,5.663,149.050
C05100=1191.586,-29.903,-42.654,179.837,5.663,149.049
C05101=1191.581,-29.653,-42.667,179.840,5.663,149.048
C05102=1191.576,-29.404,-42.680,179.842,5.664,149.048
C05103=1191.571,-29.155,-42.692,179.844,5.664,149.047
C05104=1191.566,-28.905,-42.704,179.847,5.664,149.047
C05105=1191.561,-28.655,-42.717,179.849,5.664,149.046
C05106=1191.555,-28.405,-42.730,179.851,5.665,149.045
C05107=1191.550,-28.156,-42.743,179.854,5.665,149.045
C05108=1191.545,-27.907,-42.755,179.857,5.666,149.044
C05109=1191.540,-27.656,-42.768,179.859,5.666,149.043
C05110=1191.535,-27.407,-42.780,179.861,5.666,149.043
C05111=1191.530,-27.157,-42.793,179.864,5.667,149.042
C05112=1191.525,-26.908,-42.805,179.866,5.667,149.041
C05113=1191.520,-26.658,-42.819,179.869,5.668,149.041
C05114=1191.514,-26.408,-42.832,179.872,5.668,149.040
C05115=1191.509,-26.159,-42.844,179.873,5.668,149.040
C05116=1191.504,-25.910,-42.857,179.876,5.669,149.039
C05117=1191.500,-25.660,-42.870,179.878,5.669,149.038
C05118=1191.494,-25.410,-42.882,179.881,5.670,149.037
C05119=1191.488,-25.160,-42.895,179.884,5.670,149.037
C05120=1191.483,-24.911,-42.907,179.886,5.671,149.036
C05121=1191.479,-24.661,-42.920,179.888,5.671,149.036
C05122=1191.474,-24.411,-42.933,179.891,5.671,149.035
C05123=1191.468,-24.162,-42.946,179.893,5.672,149.034
C05124=1191.463,-23.912,-42.959,179.895,5.672,149.034
C05125=1191.458,-23.643,-42.973,179.898,5.673,149.033
C05126=1191.452,-23.373,-42.987,179.901,5.673,149.032
C05127=1191.447,-23.103,-43.000,179.903,5.674,149.032
C05128=1191.440,-22.834,-43.014,179.906,5.674,149.031
C05129=1191.436,-22.584,-43.027,179.908,5.674,149.030
C05130=1191.431,-22.334,-43.040,179.911,5.674,149.030
C05131=1191.426,-22.085,-43.053,179.914,5.675,149.029
C05132=1191.420,-21.835,-43.066,179.916,5.675,149.028
C05133=1191.415,-21.585,-43.079,179.918,5.676,149.028
C05134=1191.410,-21.336,-43.091,179.921,5.677,149.027
C05135=1191.405,-21.087,-43.104,179.923,5.676,149.026
C05136=1191.400,-20.836,-43.117,179.926,5.677,149.026
C05137=1191.395,-20.587,-43.130,179.928,5.678,149.025
C05138=1191.390,-20.338,-43.143,179.931,5.678,149.024
C05139=1191.384,-20.087,-43.156,179.933,5.678,149.024
C05140=1191.379,-19.838,-43.169,179.936,5.679,149.023
C05141=1191.374,-19.589,-43.182,179.937,5.679,149.023
C05142=1191.369,-19.339,-43.196,179.940,5.679,149.022
C05143=1191.364,-19.090,-43.208,179.943,5.680,149.021
C05144=1191.359,-18.840,-43.221,179.945,5.680,149.020
C05145=1191.354,-18.590,-43.234,179.948,5.681,149.020
C05146=1191.348,-18.341,-43.247,179.950,5.682,149.019
C05147=1191.344,-18.091,-43.260,179.952,5.681,149.019
C05148=1191.338,-17.841,-43.273,179.955,5.682,149.018
C05149=1191.333,-17.592,-43.286,179.958,5.682,149.017
C05150=1191.329,-17.342,-43.300,179.960,5.683,149.017
C05151=1191.323,-17.093,-43.313,179.963,5.684,149.016
C05152=1191.318,-16.843,-43.326,179.965,5.684,149.015
C05153=1191.313,-16.593,-43.339,179.967,5.684,149.015
C05154=1191.307,-16.344,-43.351,179.970,5.684,149.014
C05155=1191.303,-16.094,-43.365,179.972,5.685,149.014
C05156=1191.297,-15.845,-43.378,179.975,5.685,149.013
C05157=1191.293,-15.595,-43.391,179.977,5.686,149.012
C05158=1191.287,-15.345,-43.405,179.980,5.686,149.011
C05159=1191.282,-15.096,-43.417,179.982,5.687,149.011
C05160=1191.277,-14.846,-43.431,179.984,5.687,149.010
C05161=1191.272,-14.597,-43.444,179.987,5.687,149.010
C05162=1191.267,-14.347,-43.457,179.990,5.688,149.009
C05163=1191.261,-14.097,-43.470,179.992,5.688,149.008
C05164=1191.257,-13.848,-43.484,179.994,5.689,149.008
C05165=1191.251,-13.598,-43.497,179.997,5.690,149.007
C05166=1191.246,-13.349,-43.510,180.000,5.690,149.006
C05167=1191.241,-13.098,-43.523,-179.998,5.690,149.006
C05168=1191.236,-12.850,-43.537,-179.996,5.691,149.005
C05169=1191.231,-12.599,-43.550,-179.993,5.691,149.005
C05170=1191.226,-12.350,-43.563,-179.991,5.692,149.004
C05171=1191.221,-12.100,-43.577,-179.988,5.692,149.003
C05172=1191.216,-11.851,-43.590,-179.985,5.693,149.002
C05173=1191.210,-11.601,-43.603,-179.983,5.693,149.002
C05174=1191.206,-11.352,-43.616,-179.981,5.693,149.001
C05175=1191.200,-11.102,-43.630,-179.978,5.694,149.001
C05176=1191.195,-10.852,-43.643,-179.976,5.694,149.000
C05177=1191.190,-10.603,-43.657,-179.974,5.695,148.999
C05178=1191.185,-10.353,-43.669,-179.971,5.695,148.999
C05179=1191.180,-10.104,-43.684,-179.968,5.696,148.998
C05180=1191.175,-9.854,-43.696,-179.966,5.696,148.997
C05181=1191.170,-9.604,-43.710,-179.963,5.697,148.997
C05182=1191.165,-9.355,-43.723,-179.961,5.698,148.996
C05183=1191.160,-9.105,-43.737,-179.959,5.697,148.996
C05184=1191.155,-8.856,-43.750,-179.956,5.698,148.995
C05185=1191.150,-8.606,-43.764,-179.953,5.698,148.994
C05186=1191.144,-8.357,-43.776,-179.951,5.699,148.994
C05187=1191.139,-8.107,-43.791,-179.949,5.700,148.993
C05188=1191.134,-7.857,-43.804,-179.946,5.700,148.992
C05189=1191.129,-7.608,-43.817,-179.943,5.700,148.992
C05190=1191.124,-7.358,-43.831,-179.941,5.701,148.991
C05191=1191.119,-7.109,-43.844,-179.939,5.701,148.990
C05192=1191.113,-6.859,-43.858,-179.936,5.701,148.990
C05193=1191.109,-6.610,-43.872,-179.934,5.702,148.989
C05194=1191.103,-6.360,-43.884,-179.931,5.702,148.988
C05195=1191.098,-6.111,-43.899,-179.929,5.703,148.988
C05196=1191.093,-5.861,-43.911,-179.926,5.704,148.987
C05197=1191.088,-5.611,-43.926,-179.924,5.704,148.987
C05198=1191.083,-5.361,-43.939,-179.921,5.705,148.986
C05199=1191.078,-5.112,-43.952,-179.919,5.706,148.985
C05200=1191.073,-4.862,-43.966,-179.916,5.706,148.985
C05201=1191.067,-4.613,-43.980,-179.914,5.706,148.984
C05202=1191.063,-4.364,-43.994,-179.911,5.706,148.983
C05203=1191.057,-4.114,-44.007,-179.909,5.707,148.983
C05204=1191.052,-3.864,-44.021,-179.907,5.707,148.982
C05205=1191.048,-3.614,-44.034,-179.904,5.708,148.981
C05206=1191.042,-3.365,-44.048,-179.901,5.708,148.981
C05207=1191.037,-3.116,-44.062,-179.899,5.709,148.980
C05208=1191.032,-2.866,-44.075,-179.896,5.710,148.980
C05209=1191.027,-2.617,-44.089,-179.894,5.710,148.979
C05210=1191.022,-2.366,-44.103,-179.891,5.711,148.978
C05211=1191.017,-2.118,-44.116,-179.889,5.711,148.978
C05212=1191.012,-1.868,-44.130,-179.887,5.711,148.977
C05213=1191.006,-1.618,-44.143,-179.884,5.712,148.976
C05214=1191.001,-1.369,-44.158,-179.882,5.712,148.976
C05215=1190.997,-1.119,-44.171,-179.879,5.713,148.975
C05216=1190.991,-0.870,-44.185,-179.877,5.714,148.975
C05217=1190.986,-0.620,-44.199,-179.874,5.714,148.974
C05218=1190.981,-0.370,-44.213,-179.871,5.715,148.973
C05219=1190.976,-0.121,-44.226,-179.869,5.715,148.972
C05220=1190.971,0.129,-44.240,-179.867,5.716,148.972
C05221=1190.966,0.379,-44.254,-179.864,5.716,148.971
C05222=1190.961,0.628,-44.268,-179.861,5.717,148.971
C05223=1190.956,0.878,-44.282,-179.859,5.717,148.970
C05224=1190.951,1.127,-44.295,-179.856,5.718,148.969
C05225=1190.946,1.376,-44.309,-179.854,5.718,148.969
C05226=1190.941,1.626,-44.324,-179.852,5.718,148.968
C05227=1190.936,1.876,-44.337,-179.849,5.719,148.967
C05228=1190.930,2.125,-44.351,-179.847,5.719,148.967
C05229=1190.925,2.395,-44.366,-179.844,5.720,148.966
C05230=1190.920,2.664,-44.381,-179.841,5.720,148.965
C05231=1190.915,2.933,-44.396,-179.838,5.722,148.965
C05232=1190.909,3.201,-44.411,-179.836,5.722,148.964
C05233=1190.904,3.451,-44.425,-179.833,5.723,148.964
C05234=1190.899,3.702,-44.439,-179.830,5.723,148.963
C05235=1190.893,3.951,-44.453,-179.828,5.723,148.962
C05236=1190.888,4.200,-44.467,-179.826,5.724,148.961
C05237=1190.883,4.450,-44.481,-179.824,5.724,148.961
C05238=1190.879,4.699,-44.495,-179.821,5.725,148.960
C05239=1190.873,4.948,-44.509,-179.818,5.725,148.960
C05240=1190.868,5.198,-44.523,-179.816,5.726,148.959
C05241=1190.863,5.448,-44.537,-179.813,5.727,148.959
C05242=1190.858,5.698,-44.551,-179.811,5.727,148.958
C05243=1190.853,5.947,-44.565,-179.808,5.728,148.957
C05244=1190.848,6.197,-44.579,-179.806,5.728,148.956
C05245=1190.843,6.447,-44.593,-179.803,5.729,148.956
C05246=1190.837,6.696,-44.607,-179.801,5.730,148.955
C05247=1190.832,6.945,-44.622,-179.798,5.730,148.955
C05248=1190.828,7.195,-44.635,-179.795,5.730,148.954
C05249=1190.823,7.444,-44.649,-179.793,5.731,148.953
C05250=1190.818,7.694,-44.664,-179.791,5.732,148.953
C05251=1190.813,7.943,-44.678,-179.788,5.732,148.952
C05252=1190.808,8.193,-44.692,-179.785,5.733,148.951
C05253=1190.803,8.443,-44.706,-179.783,5.734,148.951
C05254=1190.798,8.692,-44.720,-179.780,5.734,148.950
C05255=1190.792,8.941,-44.734,-179.778,5.735,148.950
C05256=1190.787,9.191,-44.749,-179.775,5.735,148.949
C05257=1190.782,9.441,-44.763,-179.773,5.736,148.948
C05258=1190.777,9.690,-44.777,-179.770,5.736,148.948
C05259=1190.772,9.940,-44.792,-179.768,5.736,148.947
C05260=1190.767,10.189,-44.805,-179.766,5.737,148.946
C05261=1190.762,10.439,-44.820,-179.763,5.738,148.946
C05262=1190.757,10.689,-44.834,-179.761,5.738,148.945
C05263=1190.752,10.938,-44.848,-179.758,5.738,148.945
C05264=1190.747,11.188,-44.863,-179.756,5.739,148.944
C05265=1190.741,11.437,-44.876,-179.753,5.740,148.943
C05266=1190.736,11.687,-44.891,-179.751,5.740,148.943
C05267=1190.731,11.936,-44.905,-179.748,5.741,148.942
C05268=1190.726,12.186,-44.919,-179.745,5.741,148.941
C05269=1190.722,12.435,-44.934,-179.743,5.742,148.941
C05270=1190.717,12.685,-44.949,-179.741,5.743,148.940
C05271=1190.711,12.934,-44.962,-179.738,5.743,148.940
C05272=1190.706,13.184,-44.977,-179.735,5.744,148.939
C05273=1190.701,13.434,-44.992,-179.733,5.745,148.938
C05274=1190.696,13.683,-45.006,-179.730,5.745,148.938
C05275=1190.691,13.933,-45.020,-179.728,5.746,148.937
C05276=1190.686,14.182,-45.035,-179.725,5.746,148.936
C05277=1190.681,14.431,-45.049,-179.723,5.747,148.936
C05278=1190.676,14.681,-45.063,-179.720,5.747,148.935
C05279=1190.671,14.931,-45.078,-179.718,5.748,148.935
C05280=1190.666,15.180,-45.092,-179.715,5.748,148.934
C05281=1190.661,15.429,-45.107,-179.713,5.749,148.933
C05282=1190.656,15.679,-45.121,-179.710,5.750,148.933
C05283=1190.650,15.929,-45.136,-179.708,5.750,148.932
C05284=1190.645,16.179,-45.150,-179.705,5.751,148.932
C05285=1190.641,16.428,-45.165,-179.703,5.752,148.931
C05286=1190.635,16.677,-45.179,-179.700,5.752,148.930
C05287=1190.630,16.927,-45.193,-179.697,5.753,148.930
C05288=1190.625,17.176,-45.208,-179.695,5.753,148.929
C05289=1190.621,17.425,-45.223,-179.693,5.754,148.928
C05290=1190.615,17.675,-45.238,-179.690,5.754,148.928
C05291=1190.610,17.925,-45.252,-179.687,5.755,148.927
C05292=1190.605,18.174,-45.267,-179.685,5.756,148.927
C05293=1190.600,18.424,-45.281,-179.683,5.756,148.926
C05294=1190.595,18.674,-45.295,-179.680,5.757,148.925
C05295=1190.590,18.924,-45.310,-179.677,5.757,148.925
C05296=1190.585,19.173,-45.325,-179.675,5.758,148.924
C05297=1190.580,19.422,-45.340,-179.672,5.759,148.923
C05298=1190.576,19.672,-45.355,-179.670,5.759,148.923
C05299=1190.571,19.921,-45.369,-179.667,5.760,148.922
C05300=1190.564,20.171,-45.383,-179.664,5.761,148.922
C05301=1190.560,20.420,-45.398,-179.662,5.762,148.921
C05302=1190.555,20.669,-45.413,-179.659,5.762,148.920
C05303=1190.550,20.919,-45.427,-179.657,5.763,148.920
C05304=1190.544,21.169,-45.443,-179.654,5.764,148.919
C05305=1190.539,21.418,-45.457,-179.652,5.764,148.918
C05306=1190.535,21.667,-45.472,-179.649,5.765,148.918
C05307=1190.530,21.917,-45.486,-179.647,5.766,148.917
C05308=1190.524,22.166,-45.502,-179.644,5.766,148.917
C05309=1190.519,22.416,-45.516,-179.642,5.767,148.916
C05310=1190.514,22.666,-45.530,-179.639,5.767,148.915
C05311=1190.509,22.915,-45.546,-179.637,5.768,148.915
C05312=1190.504,23.165,-45.560,-179.634,5.768,148.914
C05313=1190.499,23.414,-45.575,-179.631,5.769,148.913
C05314=1190.494,23.664,-45.590,-179.629,5.770,148.913
C05315=1190.489,23.913,-45.605,-179.627,5.770,148.912
C05316=1190.484,24.163,-45.619,-179.624,5.771,148.912
C05317=1190.479,24.412,-45.635,-179.621,5.771,148.911
C05318=1190.474,24.662,-45.649,-179.619,5.772,148.910
C05319=1190.469,24.911,-45.664,-179.617,5.773,148.910
C05320=1190.464,25.160,-45.680,-179.614,5.773,148.909
C05321=1190.459,25.410,-45.694,-179.612,5.774,148.909
C05322=1190.454,25.659,-45.709,-179.609,5.775,148.908
C05323=1190.449,25.910,-45.724,-179.606,5.775,148.907
C05324=1190.444,26.159,-45.739,-179.603,5.776,148.907
C05325=1190.440,26.409,-45.753,-179.601,5.777,148.906
C05326=1190.434,26.658,-45.769,-179.598,5.778,148.905
C05327=1190.429,26.907,-45.784,-179.596,5.778,148.905
C05328=1190.424,27.157,-45.799,-179.593,5.779,148.904
C05329=1190.419,27.406,-45.814,-179.591,5.780,148.904
C05330=1190.414,27.656,-45.828,-179.588,5.780,148.903
C05331=1190.409,27.906,-45.844,-179.586,5.781,148.902
C05332=1190.404,28.155,-45.859,-179.584,5.781,148.902
C05333=1190.398,28.424,-45.875,-179.581,5.782,148.901
C05334=1190.393,28.693,-45.891,-179.578,5.782,148.901
C05335=1190.388,28.961,-45.908,-179.575,5.784,148.900
C05336=1190.382,29.230,-45.923,-179.572,5.784,148.899
C05337=1190.377,29.479,-45.939,-179.570,5.785,148.898
C05338=1190.372,29.729,-45.953,-179.568,5.786,148.898
C05339=1190.367,29.978,-45.969,-179.565,5.786,148.897
C05340=1190.363,30.228,-45.984,-179.562,5.787,148.897
C05341=1190.357,30.478,-45.999,-179.560,5.787,148.896
C05342=1190.352,30.727,-46.014,-179.557,5.788,148.896
C05343=1190.347,30.977,-46.030,-179.555,5.789,148.895
C05344=1190.342,31.226,-46.045,-179.552,5.790,148.894
C05345=1190.337,31.476,-46.060,-179.549,5.791,148.894
C05346=1190.332,31.725,-46.075,-179.547,5.791,148.893
C05347=1190.327,31.974,-46.090,-179.544,5.792,148.892
C05348=1190.323,32.224,-46.106,-179.542,5.792,148.892
C05349=1190.317,32.473,-46.121,-179.539,5.793,148.891
C05350=1190.312,32.723,-46.135,-179.537,5.794,148.891
C05351=1190.307,32.973,-46.151,-179.534,5.794,148.890
C05352=1190.302,33.222,-46.166,-179.532,5.795,148.889
C05353=1190.297,33.471,-46.182,-179.529,5.796,148.889
C05354=1190.293,33.721,-46.197,-179.527,5.796,148.888
C05355=1190.287,33.971,-46.212,-179.524,5.798,148.888
C05356=1190.282,34.220,-46.227,-179.521,5.798,148.887
C05357=1190.277,34.469,-46.242,-179.519,5.799,148.886
C05358=1190.272,34.719,-46.258,-179.516,5.799,148.886
C05359=1190.267,34.968,-46.273,-179.514,5.800,148.885
C05360=1190.262,35.218,-46.289,-179.511,5.801,148.885
C05361=1190.258,35.467,-46.304,-179.509,5.801,148.884
C05362=1190.252,35.716,-46.319,-179.506,5.802,148.883
C05363=1190.247,35.966,-46.335,-179.504,5.803,148.883
C05364=1190.242,36.216,-46.349,-179.500,5.804,148.882
C05365=1190.237,36.466,-46.365,-179.498,5.805,148.882
C05366=1190.232,36.715,-46.380,-179.496,5.805,148.881
C05367=1190.227,36.964,-46.396,-179.493,5.806,148.880
C05368=1190.222,37.214,-46.411,-179.490,5.806,148.880
C05369=1190.218,37.463,-46.427,-179.488,5.807,148.879
C05370=1190.212,37.713,-46.442,-179.486,5.808,148.878
C05371=1190.207,37.962,-46.458,-179.483,5.808,148.878
C05372=1190.202,38.211,-46.473,-179.481,5.809,148.877
C05373=1190.197,38.461,-46.489,-179.478,5.810,148.877
C05374=1190.192,38.711,-46.505,-179.475,5.811,148.876
C05375=1190.187,38.960,-46.520,-179.473,5.812,148.876
C05376=1190.182,39.209,-46.535,-179.470,5.812,148.875
C05377=1190.177,39.459,-46.551,-179.468,5.813,148.874
C05378=1190.172,39.709,-46.567,-179.465,5.814,148.874
C05379=1190.167,39.958,-46.582,-179.463,5.814,148.873
C05380=1190.162,40.207,-46.597,-179.459,5.816,148.872
C05381=1190.157,40.457,-46.613,-179.457,5.816,148.872
C05382=1190.153,40.706,-46.629,-179.455,5.817,148.871
C05383=1190.147,40.955,-46.644,-179.452,5.817,148.871
C05384=1190.142,41.205,-46.660,-179.450,5.818,148.870
C05385=1190.137,41.455,-46.676,-179.447,5.819,148.870
C05386=1190.132,41.704,-46.691,-179.445,5.819,148.869
C05387=1190.127,41.953,-46.707,-179.442,5.820,148.868
C05388=1190.122,42.203,-46.723,-179.439,5.822,148.868
C05389=1190.117,42.453,-46.738,-179.437,5.822,148.867
C05390=1190.111,42.702,-46.754,-179.434,5.823,148.866
C05391=1190.107,42.951,-46.769,-179.432,5.824,148.866
C05392=1190.102,43.201,-46.785,-179.429,5.824,148.865
C05393=1190.097,43.450,-46.801,-179.427,5.825,148.865
C05394=1190.092,43.699,-46.817,-179.424,5.826,148.864
C05395=1190.087,43.950,-46.833,-179.421,5.827,148.863
C05396=1190.082,44.198,-46.848,-179.419,5.827,148.863
C05397=1190.077,44.447,-46.864,-179.416,5.828,148.862
C05398=1190.072,44.698,-46.880,-179.414,5.829,148.862
C05399=1190.067,44.947,-46.895,-179.411,5.829,148.861
C05400=1190.061,45.196,-46.911,-179.409,5.830,148.861
C05401=1190.058,45.446,-46.927,-179.406,5.831,148.860
C05402=1190.052,45.695,-46.943,-179.403,5.832,148.859
C05403=1190.048,45.945,-46.959,-179.401,5.833,148.859
C05404=1190.042,46.194,-46.975,-179.398,5.833,148.858
C05405=1190.037,46.443,-46.990,-179.396,5.834,148.857
C05406=1190.032,46.693,-47.006,-179.393,5.835,148.857
C05407=1190.027,46.943,-47.022,-179.390,5.836,148.856
C05408=1190.022,47.192,-47.038,-179.388,5.837,148.856
C05409=1190.018,47.441,-47.054,-179.385,5.837,148.855
C05410=1190.012,47.691,-47.069,-179.383,5.838,148.855
C05411=1190.008,47.940,-47.086,-179.380,5.839,148.854
C05412=1190.003,48.190,-47.102,-179.378,5.839,148.853
C05413=1189.997,48.439,-47.117,-179.375,5.841,148.853
C05414=1189.993,48.688,-47.134,-179.372,5.841,148.852
C05415=1189.987,48.938,-47.149,-179.370,5.842,148.852
C05416=1189.983,49.187,-47.166,-179.367,5.843,148.851
C05417=1189.977,49.437,-47.182,-179.365,5.843,148.850
C05418=1189.973,49.687,-47.198,-179.362,5.845,148.850
C05419=1189.968,49.936,-47.214,-179.359,5.845,148.849
C05420=1189.962,50.185,-47.229,-179.357,5.846,148.849
C05421=1189.958,50.435,-47.246,-179.355,5.847,148.848
C05422=1189.952,50.684,-47.262,-179.352,5.847,148.847
C05423=1189.947,50.934,-47.278,-179.349,5.849,148.847
C05424=1189.943,51.183,-47.293,-179.347,5.850,148.846
C05425=1189.938,51.433,-47.309,-179.344,5.850,148.846
C05426=1189.933,51.681,-47.326,-179.342,5.851,148.845
C05427=1189.928,51.932,-47.342,-179.339,5.852,148.845
C05428=1189.923,52.180,-47.358,-179.336,5.853,148.844
C05429=1189.919,52.430,-47.374,-179.334,5.854,148.843
C05430=1189.914,52.679,-47.390,-179.331,5.854,148.843
C05431=1189.908,52.930,-47.407,-179.329,5.855,148.842
C05432=1189.903,53.178,-47.423,-179.326,5.856,148.842
C05433=1189.898,53.428,-47.439,-179.323,5.857,148.841
C05434=1189.893,53.677,-47.455,-179.321,5.858,148.840
C05435=1189.888,53.927,-47.471,-179.318,5.858,148.840
C05436=1189.883,54.176,-47.488,-179.316,5.859,148.839
C05437=1189.878,54.445,-47.505,-179.313,5.860,148.839
C05438=1189.873,54.713,-47.523,-179.310,5.861,148.838
C05439=1189.867,54.982,-47.540,-179.308,5.862,148.837
C05440=1189.862,55.250,-47.557,-179.305,5.863,148.837
C05441=1189.857,55.500,-47.573,-179.302,5.864,148.836
C05442=1189.852,55.749,-47.590,-179.300,5.864,148.836
C05443=1189.847,55.999,-47.606,-179.297,5.865,148.835
C05444=1189.842,56.248,-47.622,-179.294,5.866,148.834
C05445=1189.837,56.497,-47.639,-179.292,5.867,148.834
C05446=1189.832,56.747,-47.655,-179.289,5.868,148.833
C05447=1189.827,56.996,-47.671,-179.286,5.868,148.833
C05448=1189.822,57.245,-47.688,-179.284,5.869,148.832
C05449=1189.817,57.495,-47.704,-179.281,5.871,148.831
C05450=1189.812,57.745,-47.721,-179.279,5.871,148.831
C05451=1189.807,57.993,-47.737,-179.276,5.872,148.830
C05452=1189.802,58.244,-47.753,-179.274,5.872,148.830
C05453=1189.797,58.492,-47.770,-179.271,5.874,148.829
C05454=1189.793,58.742,-47.786,-179.268,5.875,148.829
C05455=1189.788,58.991,-47.802,-179.266,5.875,148.828
C05456=1189.782,59.241,-47.819,-179.264,5.876,148.828
C05457=1189.778,59.491,-47.836,-179.260,5.877,148.827
C05458=1189.773,59.739,-47.852,-179.258,5.878,148.826
C05459=1189.768,59.989,-47.869,-179.256,5.879,148.826
C05460=1189.763,60.238,-47.884,-179.253,5.879,148.825
C05461=1189.758,60.488,-47.902,-179.250,5.881,148.825
C05462=1189.753,60.737,-47.918,-179.248,5.882,148.824
C05463=1189.748,60.986,-47.934,-179.245,5.882,148.823
C05464=1189.744,61.236,-47.951,-179.243,5.883,148.823
C05465=1189.737,61.485,-47.967,-179.240,5.884,148.822
C05466=1189.733,61.735,-47.984,-179.237,5.885,148.822
C05467=1189.728,61.984,-48.001,-179.235,5.886,148.821
C05468=1189.723,62.233,-48.017,-179.232,5.886,148.820
C05469=1189.718,62.483,-48.034,-179.229,5.888,148.820
C05470=1189.714,62.732,-48.051,-179.227,5.889,148.819
C05471=1189.708,62.982,-48.067,-179.225,5.890,148.819
C05472=1189.704,63.231,-48.083,-179.222,5.890,148.818
C05473=1189.699,63.481,-48.100,-179.219,5.891,148.818
C05474=1189.694,63.730,-48.117,-179.217,5.892,148.817
C05475=1189.689,63.979,-48.133,-179.214,5.893,148.817
C05476=1189.684,64.229,-48.151,-179.212,5.894,148.816
C05477=1189.679,64.478,-48.167,-179.209,5.895,148.815
C05478=1189.674,64.727,-48.184,-179.206,5.896,148.815
C05479=1189.669,64.977,-48.201,-179.204,5.897,148.814
C05480=1189.664,65.226,-48.217,-179.201,5.898,148.814
C05481=1189.659,65.476,-48.234,-179.199,5.899,148.813
C05482=1189.654,65.725,-48.251,-179.196,5.899,148.813
C05483=1189.649,65.974,-48.267,-179.193,5.900,148.812
C05484=1189.645,66.224,-48.284,-179.191,5.902,148.811
C05485=1189.639,66.473,-48.301,-179.188,5.902,148.811
C05486=1189.634,66.722,-48.318,-179.186,5.903,148.810
C05487=1189.629,66.972,-48.335,-179.183,5.904,148.810
C05488=1189.625,67.221,-48.352,-179.180,5.905,148.809
C05489=1189.620,67.471,-48.368,-179.178,5.906,148.809
C05490=1189.614,67.720,-48.385,-179.175,5.906,148.808
C05491=1189.610,67.970,-48.402,-179.172,5.908,148.808
